C07305=1204.905,265.539,-64.446,-176.922,6.908,148.380
C07306=1204.909,265.290,-64.417,-176.924,6.905,148.380
C07307=1204.914,265.042,-64.390,-176.927,6.904,148.381
C07308=1204.918,264.794,-64.363,-176.929,6.901,148.381
C07309=1204.923,264.545,-64.336,-176.932,6.899,148.381
C07310=1204.926,264.297,-64.307,-176.935,6.896,148.381
C07311=1204.931,264.048,-64.280,-176.937,6.893,148.381
C07312=1204.936,263.800,-64.253,-176.939,6.892,148.382
C07313=1204.939,263.551,-64.225,-176.942,6.889,148.382
C07314=1204.945,263.279,-64.195,-176.945,6.887,148.382
C07315=1204.949,263.006,-64.165,-176.947,6.884,148.382
C07316=1204.954,262.734,-64.135,-176.951,6.881,148.382
C07317=1204.959,262.460,-64.105,-176.953,6.879,148.382
C07318=1204.964,262.212,-64.077,-176.956,6.876,148.383
C07319=1204.968,261.963,-64.050,-176.958,6.874,148.383
C07320=1204.972,261.715,-64.024,-176.961,6.872,148.383
C07321=1204.976,261.467,-63.995,-176.963,6.869,148.383
C07322=1204.981,261.218,-63.968,-176.966,6.867,148.383
C07323=1204.985,260.970,-63.941,-176.968,6.865,148.383
C07324=1204.990,260.721,-63.914,-176.971,6.862,148.384
C07325=1204.994,260.473,-63.886,-176.973,6.860,148.384
C07326=1204.999,260.224,-63.859,-176.977,6.858,148.384
C07327=1205.003,259.976,-63.832,-176.979,6.855,148.384
C07328=1205.008,259.727,-63.805,-176.981,6.853,148.384
C07329=1205.012,259.479,-63.777,-176.984,6.850,148.384
C07330=1205.017,259.231,-63.750,-176.986,6.848,148.384
C07331=1205.021,258.982,-63.723,-176.989,6.846,148.385
C07332=1205.026,258.733,-63.696,-176.992,6.843,148.385
C07333=1205.029,258.485,-63.669,-176.994,6.842,148.385
C07334=1205.034,258.236,-63.642,-176.996,6.839,148.385
C07335=1205.039,257.988,-63.615,-176.999,6.838,148.386
C07336=1205.043,257.740,-63.587,-177.002,6.835,148.386
C07337=1205.047,257.491,-63.560,-177.004,6.833,148.386
C07338=1205.052,257.242,-63.533,-177.006,6.830,148.386
C07339=1205.057,256.994,-63.506,-177.010,6.828,148.386
C07340=1205.060,256.746,-63.479,-177.012,6.826,148.386
C07341=1205.065,256.497,-63.452,-177.014,6.824,148.387
C07342=1205.070,256.249,-63.425,-177.017,6.821,148.387
C07343=1205.074,256.000,-63.398,-177.020,6.819,148.387
C07344=1205.079,255.752,-63.371,-177.022,6.817,148.387
C07345=1205.082,255.503,-63.344,-177.025,6.814,148.387
C07346=1205.087,255.254,-63.317,-177.027,6.812,148.387
C07347=1205.092,255.006,-63.290,-177.030,6.810,148.388
C07348=1205.096,254.757,-63.263,-177.032,6.807,148.388
C07349=1205.100,254.509,-63.236,-177.035,6.805,148.388
C07350=1205.105,254.261,-63.209,-177.037,6.803,148.388
C07351=1205.110,254.012,-63.182,-177.040,6.801,148.389
C07352=1205.114,253.764,-63.155,-177.043,6.798,148.389
C07353=1205.118,253.515,-63.129,-177.045,6.796,148.389
C07354=1205.123,253.267,-63.102,-177.047,6.794,148.389
C07355=1205.127,253.018,-63.075,-177.051,6.791,148.389
C07356=1205.131,252.769,-63.049,-177.053,6.789,148.389
C07357=1205.136,252.520,-63.022,-177.055,6.787,148.390
C07358=1205.140,252.272,-62.994,-177.057,6.785,148.390
C07359=1205.144,252.024,-62.968,-177.061,6.782,148.390
C07360=1205.149,251.775,-62.941,-177.063,6.780,148.390
C07361=1205.154,251.527,-62.914,-177.065,6.778,148.390
C07362=1205.158,251.278,-62.888,-177.069,6.776,148.391
C07363=1205.163,251.029,-62.861,-177.071,6.774,148.391
C07364=1205.167,250.781,-62.834,-177.073,6.772,148.391
C07365=1205.171,250.533,-62.808,-177.076,6.770,148.391
C07366=1205.176,250.284,-62.780,-177.079,6.767,148.391
C07367=1205.181,250.035,-62.754,-177.081,6.765,148.392
C07368=1205.185,249.787,-62.728,-177.083,6.763,148.392
C07369=1205.189,249.539,-62.701,-177.086,6.761,148.392
C07370=1205.193,249.290,-62.674,-177.089,6.758,148.392
C07371=1205.198,249.041,-62.648,-177.091,6.756,148.392
C07372=1205.203,248.793,-62.621,-177.094,6.754,148.393
C07373=1205.207,248.545,-62.594,-177.097,6.751,148.393
C07374=1205.212,248.295,-62.568,-177.099,6.749,148.393
C07375=1205.216,248.047,-62.541,-177.102,6.747,148.393
C07376=1205.220,247.799,-62.514,-177.104,6.745,148.393
C07377=1205.224,247.550,-62.489,-177.107,6.742,148.394
C07378=1205.229,247.301,-62.462,-177.109,6.740,148.394
C07379=1205.233,247.053,-62.436,-177.112,6.738,148.394
C07380=1205.238,246.804,-62.409,-177.114,6.737,148.394
C07381=1205.242,246.556,-62.382,-177.117,6.733,148.394
C07382=1205.248,246.308,-62.356,-177.120,6.732,148.395
C07383=1205.251,246.059,-62.330,-177.122,6.729,148.395
C07384=1205.256,245.810,-62.304,-177.124,6.728,148.395
C07385=1205.260,245.562,-62.277,-177.128,6.725,148.395
C07386=1205.265,245.313,-62.251,-177.130,6.723,148.395
C07387=1205.269,245.065,-62.224,-177.132,6.721,148.396
C07388=1205.274,244.816,-62.198,-177.135,6.719,148.396
C07389=1205.278,244.567,-62.171,-177.137,6.717,148.396
C07390=1205.283,244.318,-62.145,-177.140,6.714,148.396
C07391=1205.287,244.070,-62.119,-177.142,6.712,148.397
C07392=1205.291,243.821,-62.093,-177.145,6.710,148.397
C07393=1205.296,243.573,-62.066,-177.147,6.708,148.397
C07394=1205.301,243.325,-62.040,-177.150,6.705,148.397
C07395=1205.305,243.076,-62.013,-177.153,6.703,148.398
C07396=1205.310,242.827,-61.988,-177.155,6.701,148.398
C07397=1205.314,242.579,-61.962,-177.158,6.699,148.398
C07398=1205.318,242.330,-61.935,-177.160,6.697,148.398
C07399=1205.323,242.081,-61.909,-177.163,6.695,148.398
C07400=1205.327,241.833,-61.883,-177.166,6.693,148.399
C07401=1205.332,241.585,-61.857,-177.168,6.691,148.399
C07402=1205.336,241.336,-61.831,-177.171,6.689,148.399
C07403=1205.341,241.087,-61.804,-177.174,6.686,148.399
C07404=1205.345,240.839,-61.778,-177.176,6.684,148.399
C07405=1205.349,240.590,-61.752,-177.179,6.682,148.400
C07406=1205.354,240.341,-61.725,-177.181,6.680,148.400
C07407=1205.359,240.093,-61.700,-177.183,6.678,148.400
C07408=1205.363,239.844,-61.674,-177.187,6.675,148.400
C07409=1205.367,239.596,-61.648,-177.189,6.673,148.401
C07410=1205.372,239.347,-61.621,-177.191,6.671,148.401
C07411=1205.376,239.098,-61.596,-177.194,6.669,148.401
C07412=1205.381,238.850,-61.570,-177.196,6.667,148.401
C07413=1205.386,238.601,-61.544,-177.199,6.665,148.402
C07414=1205.390,238.353,-61.517,-177.202,6.663,148.402
C07415=1205.394,238.104,-61.492,-177.204,6.661,148.402
C07416=1205.398,237.855,-61.466,-177.207,6.659,148.402
C07417=1205.403,237.607,-61.440,-177.209,6.657,148.403
C07418=1205.408,237.336,-61.411,-177.212,6.654,148.403
C07419=1205.413,237.064,-61.383,-177.215,6.652,148.403
C07420=1205.418,236.793,-61.355,-177.218,6.649,148.403
C07421=1205.423,236.521,-61.327,-177.220,6.648,148.404
C07422=1205.427,236.272,-61.301,-177.223,6.645,148.404
C07423=1205.431,236.024,-61.275,-177.226,6.643,148.404
C07424=1205.437,235.775,-61.249,-177.228,6.641,148.404
C07425=1205.441,235.526,-61.223,-177.231,6.639,148.404
C07426=1205.445,235.278,-61.198,-177.233,6.637,148.405
C07427=1205.450,235.029,-61.172,-177.236,6.635,148.405
C07428=1205.454,234.781,-61.146,-177.239,6.633,148.405
C07429=1205.458,234.532,-61.121,-177.241,6.630,148.405
C07430=1205.463,234.283,-61.095,-177.244,6.628,148.406
C07431=1205.468,234.035,-61.069,-177.247,6.626,148.406
C07432=1205.473,233.786,-61.043,-177.249,6.624,148.406
C07433=1205.477,233.537,-61.018,-177.251,6.622,148.407
C07434=1205.482,233.289,-60.992,-177.254,6.621,148.407
C07435=1205.486,233.040,-60.966,-177.257,6.618,148.407
C07436=1205.490,232.791,-60.941,-177.259,6.616,148.407
C07437=1205.494,232.543,-60.915,-177.262,6.614,148.408
C07438=1205.499,232.294,-60.889,-177.264,6.612,148.408
C07439=1205.503,232.046,-60.864,-177.267,6.610,148.408
C07440=1205.508,231.797,-60.838,-177.269,6.608,148.408
C07441=1205.512,231.549,-60.813,-177.273,6.605,148.409
C07442=1205.517,231.300,-60.787,-177.275,6.603,148.409
C07443=1205.521,231.051,-60.761,-177.277,6.601,148.409
C07444=1205.526,230.802,-60.736,-177.280,6.600,148.409
C07445=1205.531,230.553,-60.710,-177.282,6.597,148.409
C07446=1205.536,230.305,-60.685,-177.285,6.596,148.410
C07447=1205.540,230.056,-60.659,-177.287,6.594,148.410
C07448=1205.544,229.808,-60.633,-177.291,6.591,148.410
C07449=1205.548,229.560,-60.608,-177.293,6.589,148.410
C07450=1205.553,229.310,-60.583,-177.295,6.587,148.411
C07451=1205.557,229.062,-60.558,-177.298,6.585,148.411
C07452=1205.562,228.813,-60.532,-177.301,6.583,148.411
C07453=1205.566,228.565,-60.506,-177.303,6.581,148.412
C07454=1205.571,228.316,-60.482,-177.305,6.579,148.412
C07455=1205.575,228.067,-60.456,-177.308,6.577,148.412
C07456=1205.580,227.818,-60.430,-177.311,6.575,148.413
C07457=1205.584,227.570,-60.405,-177.313,6.573,148.413
C07458=1205.589,227.321,-60.380,-177.316,6.571,148.413
C07459=1205.594,227.073,-60.355,-177.319,6.569,148.413
C07460=1205.598,226.824,-60.329,-177.321,6.567,148.414
C07461=1205.603,226.575,-60.304,-177.323,6.565,148.414
C07462=1205.607,226.326,-60.278,-177.326,6.563,148.414
C07463=1205.612,226.078,-60.253,-177.329,6.560,148.414
C07464=1205.616,225.829,-60.229,-177.332,6.559,148.415
C07465=1205.620,225.580,-60.203,-177.334,6.556,148.415
C07466=1205.625,225.332,-60.178,-177.337,6.555,148.415
C07467=1205.630,225.083,-60.152,-177.339,6.553,148.415
C07468=1205.634,224.835,-60.127,-177.342,6.551,148.416
C07469=1205.639,224.585,-60.102,-177.344,6.549,148.416
C07470=1205.643,224.337,-60.077,-177.347,6.547,148.416
C07471=1205.648,224.088,-60.052,-177.349,6.545,148.417
C07472=1205.652,223.840,-60.027,-177.353,6.542,148.417
C07473=1205.657,223.591,-60.002,-177.355,6.540,148.417
C07474=1205.662,223.342,-59.976,-177.357,6.538,148.417
C07475=1205.666,223.093,-59.951,-177.360,6.537,148.418
C07476=1205.670,222.845,-59.926,-177.363,6.535,148.418
C07477=1205.675,222.596,-59.901,-177.365,6.533,148.418
C07478=1205.680,222.348,-59.876,-177.368,6.531,148.418
C07479=1205.684,222.098,-59.851,-177.370,6.529,148.419
C07480=1205.688,221.850,-59.826,-177.373,6.527,148.419
C07481=1205.693,221.601,-59.801,-177.375,6.525,148.419
C07482=1205.698,221.353,-59.776,-177.379,6.523,148.420
C07483=1205.702,221.103,-59.751,-177.381,6.520,148.420
C07484=1205.706,220.856,-59.726,-177.383,6.519,148.420
C07485=1205.711,220.606,-59.701,-177.386,6.517,148.420
C07486=1205.716,220.358,-59.676,-177.389,6.515,148.421
C07487=1205.719,220.109,-59.651,-177.391,6.513,148.421
C07488=1205.725,219.860,-59.626,-177.393,6.511,148.421
C07489=1205.729,219.611,-59.601,-177.396,6.509,148.421
C07490=1205.733,219.363,-59.577,-177.399,6.507,148.422
C07491=1205.738,219.114,-59.552,-177.401,6.505,148.422
C07492=1205.743,218.865,-59.527,-177.405,6.503,148.422
C07493=1205.747,218.617,-59.502,-177.407,6.501,148.423
C07494=1205.752,218.368,-59.477,-177.409,6.499,148.423
C07495=1205.757,218.119,-59.452,-177.412,6.497,148.423
C07496=1205.760,217.871,-59.427,-177.415,6.495,148.424
C07497=1205.765,217.622,-59.403,-177.417,6.493,148.424
C07498=1205.770,217.373,-59.378,-177.420,6.491,148.424
C07499=1205.774,217.124,-59.353,-177.423,6.489,148.425
C07500=1205.779,216.876,-59.328,-177.425,6.487,148.425
C07501=1205.783,216.627,-59.304,-177.427,6.485,148.425
C07502=1205.788,216.378,-59.279,-177.430,6.484,148.425
C07503=1205.793,216.129,-59.254,-177.433,6.482,148.426
C07504=1205.797,215.880,-59.230,-177.435,6.480,148.426
C07505=1205.802,215.632,-59.204,-177.439,6.477,148.426
C07506=1205.806,215.384,-59.180,-177.441,6.475,148.426
C07507=1205.811,215.134,-59.155,-177.443,6.473,148.427
C07508=1205.815,214.886,-59.131,-177.446,6.471,148.427
C07509=1205.820,214.636,-59.106,-177.449,6.470,148.427
C07510=1205.824,214.388,-59.082,-177.451,6.468,148.428
C07511=1205.829,214.139,-59.058,-177.454,6.466,148.428
C07512=1205.833,213.890,-59.033,-177.457,6.464,148.428
C07513=1205.838,213.642,-59.008,-177.459,6.462,148.429
C07514=1205.842,213.394,-58.984,-177.461,6.460,148.429
C07515=1205.847,213.144,-58.959,-177.464,6.458,148.429
C07516=1205.851,212.896,-58.935,-177.467,6.456,148.430
C07517=1205.856,212.647,-58.910,-177.469,6.455,148.430
C07518=1205.861,212.399,-58.886,-177.472,6.453,148.430
C07519=1205.865,212.149,-58.861,-177.475,6.451,148.431
C07520=1205.869,211.901,-58.837,-177.477,6.449,148.431
C07521=1205.875,211.652,-58.812,-177.480,6.446,148.431
C07522=1205.879,211.381,-58.785,-177.483,6.444,148.431
C07523=1205.884,211.111,-58.760,-177.485,6.443,148.432
C07524=1205.889,210.841,-58.733,-177.488,6.441,148.432
C07525=1205.894,210.570,-58.706,-177.492,6.438,148.432
C07526=1205.898,210.321,-58.682,-177.494,6.436,148.433
C07527=1205.903,210.073,-58.657,-177.496,6.434,148.433
C07528=1205.907,209.824,-58.633,-177.499,6.433,148.433
C07529=1205.913,209.575,-58.608,-177.502,6.431,148.434
C07530=1205.917,209.326,-58.585,-177.504,6.429,148.434
C07531=1205.921,209.077,-58.560,-177.507,6.427,148.434
C07532=1205.926,208.829,-58.536,-177.510,6.425,148.435
C07533=1205.931,208.580,-58.512,-177.512,6.423,148.435
C07534=1205.935,208.332,-58.488,-177.515,6.422,148.435
C07535=1205.940,208.082,-58.463,-177.518,6.420,148.436
C07536=1205.944,207.834,-58.439,-177.520,6.418,148.436
C07537=1205.949,207.585,-58.415,-177.522,6.416,148.436
C07538=1205.954,207.336,-58.390,-177.525,6.414,148.436
C07539=1205.958,207.087,-58.366,-177.528,6.412,148.437
C07540=1205.962,206.839,-58.342,-177.530,6.410,148.437
C07541=1205.967,206.589,-58.318,-177.533,6.408,148.437
C07542=1205.972,206.341,-58.294,-177.536,6.407,148.438
C07543=1205.976,206.092,-58.270,-177.538,6.405,148.438
C07544=1205.981,205.843,-58.245,-177.541,6.403,148.438
C07545=1205.985,205.594,-58.221,-177.544,6.401,148.439
C07546=1205.990,205.346,-58.197,-177.546,6.399,148.439
C07547=1205.994,205.097,-58.173,-177.548,6.397,148.439
C07548=1205.999,204.848,-58.149,-177.551,6.395,148.440
C07549=1206.004,204.599,-58.125,-177.554,6.393,148.440
C07550=1206.008,204.350,-58.101,-177.556,6.392,148.440
C07551=1206.012,204.102,-58.077,-177.559,6.390,148.441
C07552=1206.017,203.853,-58.053,-177.562,6.388,148.441
C07553=1206.022,203.604,-58.029,-177.564,6.386,148.441
C07554=1206.027,203.355,-58.005,-177.567,6.384,148.442
C07555=1206.031,203.107,-57.981,-177.570,6.382,148.442
C07556=1206.036,202.858,-57.957,-177.572,6.381,148.442
C07557=1206.040,202.609,-57.934,-177.575,6.379,148.443
C07558=1206.045,202.360,-57.909,-177.577,6.377,148.443
C07559=1206.049,202.111,-57.885,-177.580,6.375,148.443
C07560=1206.054,201.862,-57.861,-177.583,6.373,148.444
C07561=1206.058,201.614,-57.837,-177.585,6.372,148.444
C07562=1206.063,201.365,-57.814,-177.588,6.369,148.444
C07563=1206.067,201.117,-57.790,-177.590,6.368,148.444
C07564=1206.072,200.868,-57.767,-177.593,6.366,148.445
C07565=1206.077,200.619,-57.742,-177.596,6.364,148.445
C07566=1206.081,200.369,-57.718,-177.598,6.362,148.446
C07567=1206.086,200.121,-57.694,-177.601,6.360,148.446
C07568=1206.090,199.872,-57.671,-177.603,6.358,148.446
C07569=1206.095,199.623,-57.647,-177.606,6.357,148.447
C07570=1206.099,199.374,-57.623,-177.609,6.355,148.447
C07571=1206.104,199.125,-57.600,-177.611,6.353,148.447
C07572=1206.109,198.877,-57.576,-177.614,6.351,148.448
C07573=1206.113,198.628,-57.552,-177.617,6.349,148.448
C07574=1206.118,198.379,-57.528,-177.619,6.347,148.448
C07575=1206.122,198.130,-57.505,-177.622,6.346,148.449
C07576=1206.127,197.881,-57.482,-177.625,6.344,148.449
C07577=1206.131,197.633,-57.458,-177.627,6.342,148.449
C07578=1206.136,197.384,-57.434,-177.629,6.341,148.450
C07579=1206.141,197.135,-57.411,-177.632,6.339,148.450
C07580=1206.145,196.886,-57.387,-177.635,6.337,148.450
C07581=1206.150,196.637,-57.363,-177.637,6.336,148.451
C07582=1206.155,196.388,-57.340,-177.640,6.334,148.451
C07583=1206.159,196.140,-57.316,-177.643,6.332,148.451
C07584=1206.164,195.891,-57.293,-177.645,6.330,148.452
C07585=1206.168,195.642,-57.269,-177.648,6.328,148.452
C07586=1206.173,195.393,-57.245,-177.651,6.326,148.452
C07587=1206.178,195.144,-57.222,-177.653,6.325,148.453
C07588=1206.182,194.895,-57.199,-177.656,6.323,148.453
C07589=1206.187,194.646,-57.175,-177.659,6.321,148.453
C07590=1206.191,194.398,-57.151,-177.661,6.319,148.454
C07591=1206.196,194.149,-57.128,-177.664,6.317,148.454
C07592=1206.201,193.900,-57.104,-177.667,6.316,148.455
C07593=1206.205,193.651,-57.081,-177.669,6.314,148.455
C07594=1206.210,193.402,-57.058,-177.671,6.313,148.455
C07595=1206.215,193.153,-57.034,-177.674,6.311,148.456
C07596=1206.219,192.904,-57.010,-177.677,6.309,148.456
C07597=1206.223,192.656,-56.987,-177.679,6.307,148.456
C07598=1206.228,192.407,-56.964,-177.682,6.305,148.457
C07599=1206.233,192.157,-56.941,-177.685,6.304,148.457
C07600=1206.237,191.908,-56.917,-177.687,6.302,148.457
C07601=1206.242,191.659,-56.894,-177.690,6.300,148.458
C07602=1206.247,191.410,-56.871,-177.693,6.298,148.458
C07603=1206.252,191.163,-56.847,-177.695,6.296,148.458
C07604=1206.256,190.914,-56.824,-177.698,6.295,148.459
C07605=1206.260,190.665,-56.801,-177.700,6.293,148.459
C07606=1206.265,190.416,-56.777,-177.703,6.292,148.459
C07607=1206.270,190.167,-56.754,-177.705,6.290,148.460
C07608=1206.274,189.918,-56.731,-177.708,6.288,148.460
C07609=1206.279,189.669,-56.707,-177.711,6.286,148.461
C07610=1206.283,189.420,-56.685,-177.713,6.284,148.461
C07611=1206.288,189.171,-56.661,-177.716,6.283,148.461
C07612=1206.293,188.923,-56.638,-177.718,6.281,148.462
C07613=1206.298,188.674,-56.615,-177.721,6.279,148.462
C07614=1206.302,188.425,-56.592,-177.724,6.277,148.462
C07615=1206.306,188.176,-56.569,-177.726,6.276,148.463
C07616=1206.311,187.927,-56.545,-177.729,6.274,148.463
C07617=1206.316,187.678,-56.522,-177.731,6.273,148.463
C07618=1206.320,187.429,-56.499,-177.734,6.271,148.464
C07619=1206.325,187.181,-56.476,-177.737,6.269,148.464
C07620=1206.330,186.931,-56.454,-177.739,6.267,148.464
C07621=1206.335,186.682,-56.430,-177.742,6.265,148.465
C07622=1206.339,186.433,-56.408,-177.744,6.263,148.465
C07623=1206.343,186.184,-56.384,-177.747,6.262,148.465
C07624=1206.348,185.935,-56.361,-177.749,6.261,148.466
C07625=1206.353,185.687,-56.338,-177.752,6.259,148.466
C07626=1206.358,185.418,-56.313,-177.755,6.257,148.467
C07627=1206.363,185.148,-56.288,-177.758,6.256,148.467
C07628=1206.368,184.878,-56.264,-177.761,6.253,148.467
C07629=1206.373,184.609,-56.239,-177.764,6.251,148.468
C07630=1206.377,184.360,-56.216,-177.766,6.249,148.468
C07631=1206.382,184.111,-56.193,-177.768,6.248,148.469
C07632=1206.387,183.861,-56.170,-177.771,6.246,148.469
C07633=1206.391,183.612,-56.147,-177.774,6.245,148.469
C07634=1206.396,183.364,-56.124,-177.777,6.243,148.470
C07635=1206.401,183.115,-56.101,-177.779,6.241,148.470
C07636=1206.405,182.866,-56.079,-177.782,6.240,148.471
C07637=1206.410,182.617,-56.056,-177.785,6.238,148.471
C07638=1206.414,182.368,-56.033,-177.787,6.237,148.471
C07639=1206.419,182.120,-56.010,-177.790,6.235,148.472
C07640=1206.423,181.870,-55.988,-177.792,6.233,148.472
C07641=1206.428,181.621,-55.964,-177.795,6.231,148.472
C07642=1206.433,181.372,-55.941,-177.797,6.229,148.473
C07643=1206.438,181.124,-55.919,-177.800,6.228,148.473
C07644=1206.442,180.875,-55.896,-177.802,6.227,148.473
C07645=1206.446,180.626,-55.873,-177.805,6.225,148.474
C07646=1206.452,180.377,-55.851,-177.808,6.223,148.474
C07647=1206.456,180.128,-55.828,-177.811,6.222,148.475
C07648=1206.461,179.879,-55.806,-177.813,6.220,148.475
C07649=1206.465,179.630,-55.783,-177.816,6.218,148.475
C07650=1206.470,179.381,-55.760,-177.818,6.217,148.476
C07651=1206.474,179.132,-55.738,-177.821,6.215,148.476
C07652=1206.479,178.883,-55.714,-177.823,6.213,148.477
C07653=1206.484,178.634,-55.693,-177.826,6.212,148.477
C07654=1206.489,178.385,-55.669,-177.829,6.210,148.477
C07655=1206.493,178.136,-55.647,-177.831,6.208,148.478
C07656=1206.498,177.888,-55.624,-177.834,6.207,148.478
C07657=1206.503,177.638,-55.602,-177.837,6.205,148.479
C07658=1206.507,177.390,-55.580,-177.839,6.204,148.479
C07659=1206.512,177.141,-55.557,-177.842,6.202,148.479
C07660=1206.516,176.892,-55.535,-177.845,6.200,148.480
C07661=1206.521,176.642,-55.512,-177.847,6.198,148.480
C07662=1206.526,176.394,-55.489,-177.849,6.197,148.480
C07663=1206.531,176.145,-55.467,-177.852,6.195,148.481
C07664=1206.535,175.896,-55.444,-177.855,6.194,148.481
C07665=1206.540,175.647,-55.422,-177.857,6.192,148.481
C07666=1206.545,175.398,-55.400,-177.861,6.190,148.482
C07667=1206.548,175.149,-55.377,-177.863,6.189,148.482
C07668=1206.554,174.900,-55.355,-177.865,6.188,148.483
C07669=1206.558,174.651,-55.332,-177.868,6.186,148.483
C07670=1206.563,174.403,-55.310,-177.871,6.184,148.484
C07671=1206.568,174.153,-55.288,-177.873,6.182,148.484
C07672=1206.572,173.904,-55.265,-177.875,6.181,148.484
C07673=1206.577,173.656,-55.243,-177.878,6.179,148.485
C07674=1206.582,173.406,-55.221,-177.881,6.178,148.485
C07675=1206.586,173.158,-55.198,-177.884,6.176,148.486
C07676=1206.591,172.909,-55.176,-177.887,6.174,148.486
C07677=1206.596,172.659,-55.153,-177.889,6.173,148.486
C07678=1206.600,172.411,-55.131,-177.891,6.171,148.487
C07679=1206.604,172.162,-55.109,-177.894,6.170,148.487
C07680=1206.609,171.913,-55.087,-177.897,6.168,148.487
C07681=1206.614,171.663,-55.065,-177.899,6.167,148.488
C07682=1206.619,171.415,-55.042,-177.902,6.165,148.488
C07683=1206.623,171.166,-55.020,-177.905,6.164,148.489
C07684=1206.628,170.916,-54.998,-177.907,6.162,148.489
C07685=1206.633,170.668,-54.976,-177.910,6.160,148.489
C07686=1206.637,170.418,-54.954,-177.912,6.159,148.490
C07687=1206.642,170.170,-54.931,-177.915,6.157,148.490
C07688=1206.647,169.921,-54.909,-177.918,6.156,148.491
C07689=1206.652,169.672,-54.887,-177.920,6.154,148.491
C07690=1206.656,169.423,-54.865,-177.923,6.153,148.492
C07691=1206.661,169.174,-54.843,-177.925,6.151,148.492
C07692=1206.665,168.925,-54.821,-177.928,6.149,148.492
C07693=1206.670,168.676,-54.798,-177.931,6.148,148.493
C07694=1206.675,168.427,-54.776,-177.933,6.147,148.493
C07695=1206.680,168.178,-54.755,-177.936,6.145,148.494
C07696=1206.684,167.929,-54.733,-177.938,6.143,148.494
C07697=1206.689,167.680,-54.711,-177.941,6.141,148.494
C07698=1206.693,167.431,-54.689,-177.943,6.140,148.495
C07699=1206.699,167.182,-54.667,-177.946,6.139,148.495
C07700=1206.703,166.933,-54.644,-177.949,6.137,148.495
C07701=1206.708,166.684,-54.623,-177.952,6.135,148.496
C07702=1206.712,166.435,-54.601,-177.954,6.134,148.496
C07703=1206.717,166.186,-54.579,-177.956,6.133,148.497
C07704=1206.721,165.937,-54.557,-177.959,6.131,148.497
C07705=1206.726,165.688,-54.535,-177.962,6.129,148.498
C07706=1206.730,165.439,-54.513,-177.964,6.128,148.498
C07707=1206.736,165.190,-54.491,-177.967,6.127,148.499
C07708=1206.741,164.941,-54.469,-177.970,6.125,148.499
C07709=1206.745,164.692,-54.447,-177.972,6.123,148.499
C07710=1206.750,164.443,-54.426,-177.975,6.122,148.500
C07711=1206.754,164.194,-54.404,-177.977,6.120,148.500
C07712=1206.759,163.945,-54.382,-177.980,6.119,148.501
C07713=1206.763,163.696,-54.360,-177.982,6.118,148.501
C07714=1206.768,163.447,-54.338,-177.985,6.116,148.501
C07715=1206.773,163.199,-54.316,-177.988,6.114,148.502
C07716=1206.777,162.949,-54.294,-177.990,6.112,148.502
C07717=1206.782,162.701,-54.273,-177.993,6.112,148.503
C07718=1206.787,162.451,-54.251,-177.996,6.110,148.503
C07719=1206.792,162.202,-54.230,-177.998,6.108,148.503
C07720=1206.796,161.953,-54.208,-178.001,6.106,148.504
C07721=1206.801,161.704,-54.186,-178.003,6.105,148.504
C07722=1206.806,161.455,-54.164,-178.006,6.104,148.505
C07723=1206.810,161.206,-54.142,-178.009,6.102,148.505
C07724=1206.815,160.957,-54.121,-178.011,6.101,148.506
C07725=1206.820,160.708,-54.100,-178.014,6.099,148.506
C07726=1206.824,160.459,-54.078,-178.017,6.098,148.507
C07727=1206.829,160.210,-54.056,-178.020,6.096,148.507
C07728=1206.834,159.961,-54.035,-178.022,6.095,148.507
C07729=1206.838,159.712,-54.013,-178.024,6.093,148.508
C07730=1206.843,159.443,-53.989,-178.027,6.092,148.508
C07731=1206.848,159.174,-53.966,-178.030,6.090,148.509
C07732=1206.853,158.905,-53.943,-178.033,6.088,148.509
C07733=1206.859,158.635,-53.920,-178.036,6.087,148.510
C07734=1206.864,158.387,-53.898,-178.038,6.086,148.510
C07735=1206.868,158.138,-53.877,-178.041,6.084,148.510
C07736=1206.873,157.889,-53.854,-178.043,6.082,148.511
C07737=1206.878,157.640,-53.834,-178.046,6.082,148.511
C07738=1206.882,157.391,-53.812,-178.049,6.080,148.512
C07739=1206.886,157.142,-53.790,-178.051,6.078,148.512
C07740=1206.891,156.893,-53.769,-178.053,6.077,148.512
C07741=1206.896,156.644,-53.748,-178.057,6.076,148.513
C07742=1206.901,156.394,-53.726,-178.059,6.074,148.513
C07743=1206.906,156.145,-53.705,-178.061,6.073,148.514
C07744=1206.911,155.897,-53.683,-178.064,6.071,148.514
C07745=1206.915,155.648,-53.663,-178.067,6.069,148.515
C07746=1206.919,155.398,-53.641,-178.069,6.069,148.515
C07747=1206.924,155.149,-53.620,-178.072,6.067,148.516
C07748=1206.929,154.901,-53.598,-178.075,6.065,148.516
C07749=1206.934,154.651,-53.577,-178.077,6.064,148.517
C07750=1206.938,154.402,-53.556,-178.080,6.063,148.517
C07751=1206.943,154.153,-53.535,-178.083,6.061,148.517
C07752=1206.948,153.904,-53.513,-178.085,6.060,148.518
C07753=1206.953,153.656,-53.491,-178.088,6.058,148.518
C07754=1206.958,153.406,-53.470,-178.091,6.056,148.519
C07755=1206.962,153.157,-53.450,-178.093,6.056,148.519
C07756=1206.967,152.908,-53.428,-178.095,6.054,148.519
C07757=1206.972,152.659,-53.407,-178.099,6.052,148.520
C07758=1206.976,152.410,-53.385,-178.101,6.051,148.520
C07759=1206.981,152.161,-53.364,-178.103,6.050,148.521
C07760=1206.986,151.912,-53.343,-178.106,6.048,148.521
C07761=1206.991,151.663,-53.322,-178.109,6.047,148.522
C07762=1206.996,151.414,-53.300,-178.111,6.045,148.522
C07763=1206.999,151.164,-53.279,-178.114,6.044,148.523
C07764=1207.005,150.915,-53.258,-178.116,6.043,148.523
C07765=1207.009,150.667,-53.237,-178.119,6.041,148.524
C07766=1207.014,150.418,-53.216,-178.122,6.039,148.524
C07767=1207.019,150.169,-53.195,-178.124,6.038,148.524
C07768=1207.023,149.919,-53.173,-178.127,6.037,148.525
C07769=1207.028,149.670,-53.153,-178.129,6.036,148.525
C07770=1207.033,149.421,-53.131,-178.132,6.034,148.526
C07771=1207.038,149.172,-53.110,-178.135,6.032,148.526
C07772=1207.042,148.923,-53.090,-178.137,6.032,148.527
C07773=1207.047,148.674,-53.069,-178.140,6.030,148.527
C07774=1207.052,148.425,-53.047,-178.143,6.028,148.527
C07775=1207.056,148.176,-53.027,-178.145,6.027,148.528
C07776=1207.061,147.926,-53.006,-178.148,6.026,148.528
C07777=1207.065,147.678,-52.985,-178.150,6.024,148.529
C07778=1207.071,147.429,-52.964,-178.153,6.023,148.529
C07779=1207.076,147.180,-52.943,-178.156,6.021,148.530
C07780=1207.080,146.931,-52.922,-178.158,6.021,148.530
C07781=1207.085,146.681,-52.900,-178.161,6.019,148.531
C07782=1207.089,146.432,-52.880,-178.164,6.017,148.531
C07783=1207.094,146.183,-52.859,-178.166,6.016,148.532
C07784=1207.099,145.934,-52.838,-178.168,6.015,148.532
C07785=1207.104,145.685,-52.817,-178.171,6.014,148.533
C07786=1207.109,145.436,-52.796,-178.174,6.012,148.533
C07787=1207.113,145.187,-52.775,-178.176,6.010,148.533
C07788=1207.118,144.938,-52.754,-178.179,6.010,148.534
C07789=1207.123,144.689,-52.734,-178.182,6.008,148.534
C07790=1207.127,144.439,-52.713,-178.184,6.007,148.535
C07791=1207.132,144.190,-52.692,-178.186,6.005,148.535
C07792=1207.137,143.941,-52.671,-178.190,6.004,148.536
C07793=1207.141,143.692,-52.651,-178.192,6.003,148.536
C07794=1207.146,143.443,-52.629,-178.194,6.001,148.537
C07795=1207.151,143.194,-52.609,-178.197,6.000,148.537
C07796=1207.156,142.945,-52.588,-178.200,5.999,148.538
C07797=1207.160,142.696,-52.568,-178.202,5.997,148.538
C07798=1207.165,142.447,-52.547,-178.205,5.996,148.539
C07799=1207.170,142.198,-52.526,-178.208,5.994,148.539
C07800=1207.174,141.949,-52.506,-178.210,5.993,148.539
C07801=1207.179,141.700,-52.485,-178.213,5.992,148.540
C07802=1207.184,141.451,-52.465,-178.216,5.990,148.540
C07803=1207.189,141.201,-52.444,-178.218,5.989,148.541
C07804=1207.193,140.953,-52.423,-178.221,5.988,148.541
C07805=1207.199,140.703,-52.402,-178.223,5.987,148.542
C07806=1207.203,140.454,-52.382,-178.226,5.985,148.542
C07807=1207.208,140.205,-52.362,-178.228,5.984,148.543
C07808=1207.213,139.956,-52.341,-178.231,5.983,148.543
C07809=1207.217,139.707,-52.320,-178.234,5.981,148.544
C07810=1207.222,139.458,-52.300,-178.236,5.980,148.544
C07811=1207.227,139.209,-52.279,-178.239,5.978,148.545
C07812=1207.232,138.959,-52.259,-178.241,5.977,148.545
C07813=1207.237,138.710,-52.238,-178.244,5.976,148.546
C07814=1207.241,138.461,-52.218,-178.246,5.975,148.546
C07815=1207.246,138.212,-52.198,-178.249,5.973,148.546
C07816=1207.251,137.963,-52.177,-178.252,5.972,148.547
C07817=1207.255,137.714,-52.156,-178.254,5.971,148.547
C07818=1207.260,137.465,-52.136,-178.257,5.969,148.548
C07819=1207.265,137.216,-52.115,-178.260,5.968,148.548
C07820=1207.270,136.966,-52.095,-178.262,5.967,148.549
C07821=1207.274,136.717,-52.075,-178.265,5.966,148.549
C07822=1207.279,136.468,-52.054,-178.268,5.964,148.550
C07823=1207.284,136.219,-52.033,-178.270,5.963,148.550
C07824=1207.288,135.970,-52.013,-178.273,5.962,148.551
C07825=1207.293,135.721,-51.993,-178.276,5.960,148.551
C07826=1207.298,135.471,-51.972,-178.278,5.959,148.552
C07827=1207.302,135.222,-51.952,-178.281,5.958,148.552
C07828=1207.307,134.973,-51.932,-178.283,5.957,148.553
C07829=1207.312,134.724,-51.912,-178.286,5.955,148.553
C07830=1207.317,134.475,-51.891,-178.288,5.954,148.554
C07831=1207.322,134.226,-51.871,-178.291,5.953,148.554
C07832=1207.326,133.977,-51.851,-178.293,5.952,148.555
C07833=1207.331,133.728,-51.831,-178.296,5.950,148.555
C07834=1207.336,133.459,-51.809,-178.299,5.949,148.556
C07835=1207.342,133.191,-51.787,-178.301,5.948,148.556
C07836=1207.346,132.922,-51.765,-178.305,5.946,148.557
C07837=1207.352,132.653,-51.743,-178.307,5.945,148.557
C07838=1207.356,132.404,-51.723,-178.310,5.944,148.558
C07839=1207.361,132.155,-51.703,-178.313,5.942,148.558
C07840=1207.366,131.906,-51.683,-178.315,5.941,148.558
C07841=1207.370,131.657,-51.663,-178.318,5.940,148.559
C07842=1207.376,131.407,-51.642,-178.320,5.939,148.559
C07843=1207.380,131.158,-51.622,-178.323,5.937,148.560
C07844=1207.385,130.909,-51.602,-178.325,5.936,148.560
C07845=1207.389,130.660,-51.582,-178.328,5.935,148.561
C07846=1207.394,130.412,-51.562,-178.331,5.934,148.562
C07847=1207.399,130.162,-51.542,-178.333,5.932,148.562
C07848=1207.404,129.913,-51.521,-178.336,5.931,148.562
C07849=1207.409,129.663,-51.502,-178.339,5.930,148.563
C07850=1207.413,129.414,-51.481,-178.341,5.928,148.563
C07851=1207.419,129.165,-51.462,-178.344,5.927,148.564
C07852=1207.423,128.916,-51.442,-178.347,5.926,148.564
C07853=1207.428,128.667,-51.422,-178.349,5.925,148.565
C07854=1207.432,128.418,-51.402,-178.352,5.923,148.565
C07855=1207.437,128.168,-51.382,-178.354,5.922,148.566
C07856=1207.442,127.919,-51.362,-178.357,5.921,148.566
C07857=1207.447,127.670,-51.342,-178.359,5.920,148.567
C07858=1207.451,127.421,-51.322,-178.362,5.919,148.567
C07859=1207.456,127.172,-51.302,-178.365,5.918,148.568
C07860=1207.461,126.923,-51.282,-178.367,5.916,148.568
C07861=1207.465,126.673,-51.262,-178.370,5.915,148.569
C07862=1207.470,126.425,-51.242,-178.372,5.913,148.569
C07863=1207.476,126.175,-51.222,-178.375,5.913,148.570
C07864=1207.481,125.926,-51.202,-178.377,5.912,148.570
C07865=1207.485,125.677,-51.182,-178.380,5.910,148.571
C07866=1207.490,125.428,-51.163,-178.383,5.909,148.571
C07867=1207.495,125.178,-51.143,-178.385,5.908,148.572
C07868=1207.500,124.929,-51.123,-178.388,5.907,148.572
C07869=1207.504,124.680,-51.104,-178.390,5.905,148.573
C07870=1207.509,124.431,-51.084,-178.393,5.905,148.573
C07871=1207.513,124.182,-51.064,-178.396,5.903,148.574
C07872=1207.518,123.933,-51.044,-178.398,5.902,148.574
C07873=1207.523,123.683,-51.025,-178.401,5.901,148.575
C07874=1207.528,123.435,-51.005,-178.403,5.900,148.575
C07875=1207.533,123.185,-50.985,-178.406,5.898,148.576
C07876=1207.537,122.936,-50.965,-178.408,5.897,148.576
C07877=1207.542,122.688,-50.945,-178.412,5.896,148.577
C07878=1207.547,122.438,-50.926,-178.414,5.895,148.577
C07879=1207.552,122.188,-50.906,-178.417,5.893,148.578
C07880=1207.557,121.939,-50.886,-178.419,5.892,148.578
C07881=1207.562,121.691,-50.866,-178.422,5.891,148.579
C07882=1207.566,121.441,-50.847,-178.424,5.890,148.579
C07883=1207.571,121.191,-50.827,-178.427,5.889,148.580
C07884=1207.576,120.943,-50.808,-178.430,5.888,148.580
C07885=1207.580,120.693,-50.789,-178.432,5.887,148.581
C07886=1207.585,120.444,-50.768,-178.435,5.885,148.581
C07887=1207.590,120.196,-50.749,-178.437,5.884,148.582
C07888=1207.595,119.946,-50.729,-178.440,5.883,148.582
C07889=1207.600,119.696,-50.710,-178.442,5.882,148.583
C07890=1207.605,119.448,-50.690,-178.446,5.881,148.583
C07891=1207.609,119.198,-50.671,-178.448,5.880,148.584
C07892=1207.614,118.949,-50.652,-178.450,5.879,148.584
C07893=1207.619,118.700,-50.632,-178.453,5.877,148.585
C07894=1207.624,118.451,-50.612,-178.455,5.876,148.585
C07895=1207.628,118.201,-50.592,-178.458,5.875,148.586
C07896=1207.634,117.952,-50.573,-178.460,5.874,148.586
C07897=1207.638,117.703,-50.554,-178.464,5.873,148.587
C07898=1207.643,117.454,-50.535,-178.466,5.872,148.587
C07899=1207.648,117.205,-50.515,-178.469,5.870,148.588
C07900=1207.653,116.955,-50.496,-178.471,5.869,148.588
C07901=1207.657,116.707,-50.477,-178.474,5.869,148.589
C07902=1207.662,116.457,-50.457,-178.476,5.867,148.589
C07903=1207.667,116.208,-50.438,-178.479,5.866,148.590
C07904=1207.672,115.959,-50.418,-178.482,5.864,148.590
C07905=1207.676,115.709,-50.399,-178.484,5.864,148.591
C07906=1207.681,115.460,-50.380,-178.487,5.862,148.591
C07907=1207.686,115.211,-50.360,-178.490,5.861,148.592
C07908=1207.691,114.962,-50.341,-178.492,5.861,148.593
C07909=1207.695,114.713,-50.322,-178.494,5.859,148.593
C07910=1207.700,114.463,-50.302,-178.497,5.858,148.594
C07911=1207.706,114.214,-50.283,-178.500,5.856,148.594
C07912=1207.710,113.965,-50.263,-178.502,5.856,148.595
C07913=1207.715,113.716,-50.245,-178.504,5.855,148.595
C07914=1207.720,113.467,-50.225,-178.508,5.853,148.596
C07915=1207.725,113.218,-50.206,-178.510,5.852,148.596
C07916=1207.729,112.969,-50.187,-178.513,5.851,148.597
C07917=1207.735,112.719,-50.168,-178.515,5.850,148.597
C07918=1207.739,112.469,-50.148,-178.518,5.849,148.598
C07919=1207.744,112.221,-50.130,-178.520,5.848,148.598
C07920=1207.749,111.971,-50.110,-178.523,5.847,148.599
C07921=1207.753,111.722,-50.090,-178.526,5.845,148.599
C07922=1207.758,111.473,-50.072,-178.528,5.845,148.600
C07923=1207.763,111.224,-50.052,-178.531,5.843,148.600
C07924=1207.768,110.974,-50.034,-178.534,5.842,148.601
C07925=1207.772,110.725,-50.014,-178.536,5.841,148.601
C07926=1207.778,110.476,-49.995,-178.539,5.840,148.602
C07927=1207.782,110.227,-49.976,-178.541,5.839,148.602
C07928=1207.787,109.978,-49.957,-178.544,5.839,148.603
C07929=1207.791,109.728,-49.938,-178.546,5.837,148.603
C07930=1207.797,109.479,-49.919,-178.549,5.836,148.604
C07931=1207.802,109.230,-49.899,-178.552,5.834,148.604
C07932=1207.806,108.981,-49.881,-178.554,5.834,148.605
C07933=1207.811,108.731,-49.862,-178.556,5.833,148.605
C07934=1207.816,108.482,-49.843,-178.560,5.831,148.606
C07935=1207.821,108.233,-49.824,-178.562,5.831,148.607
C07936=1207.825,107.984,-49.805,-178.565,5.829,148.607
C07937=1207.831,107.735,-49.786,-178.567,5.829,148.608
C07938=1207.836,107.466,-49.765,-178.570,5.828,148.608
C07939=1207.841,107.198,-49.746,-178.573,5.826,148.609
C07940=1207.846,106.929,-49.725,-178.576,5.825,148.609
C07941=1207.852,106.661,-49.705,-178.578,5.824,148.610
C07942=1207.856,106.412,-49.686,-178.581,5.823,148.611
C07943=1207.861,106.162,-49.666,-178.583,5.821,148.611
C07944=1207.866,105.913,-49.648,-178.586,5.821,148.612
C07945=1207.871,105.664,-49.629,-178.589,5.819,148.612
C07946=1207.875,105.415,-49.610,-178.591,5.818,148.613
C07947=1207.880,105.165,-49.591,-178.594,5.818,148.613
C07948=1207.885,104.916,-49.572,-178.597,5.816,148.614
C07949=1207.890,104.667,-49.554,-178.599,5.816,148.614
C07950=1207.894,104.418,-49.535,-178.601,5.815,148.615
C07951=1207.899,104.169,-49.517,-178.605,5.813,148.615
C07952=1207.904,103.919,-49.497,-178.607,5.812,148.616
C07953=1207.909,103.670,-49.478,-178.609,5.812,148.616
C07954=1207.914,103.421,-49.460,-178.612,5.810,148.617
C07955=1207.918,103.172,-49.441,-178.615,5.809,148.617
C07956=1207.924,102.922,-49.422,-178.617,5.808,148.618
C07957=1207.928,102.673,-49.403,-178.620,5.807,148.619
C07958=1207.933,102.424,-49.385,-178.623,5.806,148.619
C07959=1207.938,102.175,-49.366,-178.625,5.805,148.620
C07960=1207.943,101.925,-49.347,-178.628,5.804,148.620
C07961=1207.948,101.676,-49.328,-178.630,5.803,148.621
C07962=1207.953,101.427,-49.310,-178.633,5.802,148.621
C07963=1207.957,101.177,-49.292,-178.635,5.801,148.622
C07964=1207.962,100.928,-49.272,-178.638,5.800,148.622
C07965=1207.967,100.679,-49.254,-178.641,5.798,148.623
C07966=1207.971,100.430,-49.235,-178.643,5.798,148.623
C07967=1207.977,100.180,-49.217,-178.646,5.797,148.624
C07968=1207.982,99.932,-49.198,-178.649,5.795,148.624
C07969=1207.986,99.682,-49.180,-178.651,5.795,148.625
C07970=1207.992,99.432,-49.161,-178.653,5.794,148.626
C07971=1207.996,99.184,-49.143,-178.656,5.793,148.626
C07972=1208.001,98.934,-49.124,-178.659,5.792,148.627
C07973=1208.006,98.684,-49.106,-178.661,5.791,148.627
C07974=1208.011,98.436,-49.087,-178.664,5.789,148.628
C07975=1208.015,98.186,-49.069,-178.667,5.789,148.628
C07976=1208.020,97.937,-49.051,-178.669,5.788,148.629
C07977=1208.025,97.688,-49.031,-178.671,5.787,148.629
C07978=1208.030,97.439,-49.013,-178.674,5.786,148.630
C07979=1208.035,97.189,-48.995,-178.677,5.785,148.630
C07980=1208.040,96.940,-48.976,-178.679,5.784,148.631
C07981=1208.045,96.691,-48.958,-178.682,5.782,148.631
C07982=1208.049,96.441,-48.939,-178.685,5.782,148.632
C07983=1208.054,96.192,-48.921,-178.687,5.781,148.633
C07984=1208.059,95.943,-48.903,-178.690,5.780,148.633
C07985=1208.064,95.694,-48.884,-178.692,5.779,148.634
C07986=1208.069,95.444,-48.866,-178.695,5.778,148.634
C07987=1208.074,95.195,-48.848,-178.698,5.777,148.635
C07988=1208.078,94.946,-48.829,-178.700,5.776,148.636
C07989=1208.084,94.697,-48.811,-178.703,5.775,148.636
C07990=1208.088,94.447,-48.792,-178.705,5.775,148.637
C07991=1208.093,94.198,-48.774,-178.708,5.773,148.637
C07992=1208.098,93.948,-48.756,-178.710,5.772,148.638
C07993=1208.103,93.700,-48.738,-178.713,5.771,148.638
C07994=1208.107,93.450,-48.719,-178.716,5.770,148.639
C07995=1208.113,93.201,-48.701,-178.718,5.769,148.639
C07996=1208.117,92.951,-48.683,-178.721,5.768,148.640
C07997=1208.122,92.702,-48.665,-178.724,5.767,148.640
C07998=1208.127,92.453,-48.647,-178.726,5.766,148.641
C07999=1208.132,92.203,-48.628,-178.729,5.765,148.641
C08000=1208.136,91.954,-48.610,-178.731,5.765,148.642
C08001=1208.141,91.705,-48.592,-178.734,5.763,148.643
C08002=1208.147,91.456,-48.573,-178.736,5.763,148.643
C08003=1208.152,91.207,-48.555,-178.739,5.762,148.644
C08004=1208.156,90.957,-48.537,-178.741,5.761,148.644
C08005=1208.161,90.708,-48.519,-178.744,5.760,148.645
C08006=1208.166,90.458,-48.501,-178.747,5.759,148.645
C08007=1208.171,90.209,-48.483,-178.749,5.758,148.646
C08008=1208.176,89.960,-48.465,-178.752,5.756,148.646
C08009=1208.181,89.711,-48.447,-178.754,5.756,148.647
C08010=1208.185,89.461,-48.428,-178.757,5.755,148.648
C08011=1208.190,89.212,-48.410,-178.759,5.754,148.648
C08012=1208.195,88.963,-48.393,-178.762,5.753,148.649
C08013=1208.200,88.714,-48.375,-178.765,5.752,148.649
C08014=1208.204,88.464,-48.357,-178.767,5.751,148.650
C08015=1208.209,88.215,-48.339,-178.770,5.751,148.651
C08016=1208.214,87.966,-48.321,-178.773,5.749,148.651
C08017=1208.219,87.716,-48.302,-178.775,5.748,148.652
C08018=1208.224,87.467,-48.284,-178.778,5.748,148.652
C08019=1208.228,87.218,-48.266,-178.780,5.747,148.653
C08020=1208.233,86.969,-48.248,-178.783,5.746,148.653
C08021=1208.238,86.719,-48.230,-178.785,5.745,148.654
C08022=1208.243,86.470,-48.213,-178.788,5.744,148.654
C08023=1208.248,86.220,-48.195,-178.791,5.743,148.655
C08024=1208.253,85.971,-48.177,-178.793,5.742,148.655
C08025=1208.258,85.722,-48.159,-178.796,5.741,148.656
C08026=1208.263,85.473,-48.141,-178.798,5.741,148.657
C08027=1208.267,85.223,-48.123,-178.801,5.739,148.657
C08028=1208.272,84.974,-48.105,-178.804,5.738,148.658
C08029=1208.277,84.725,-48.087,-178.806,5.737,148.658
C08030=1208.282,84.475,-48.070,-178.809,5.737,148.659
C08031=1208.287,84.226,-48.052,-178.811,5.736,148.660
C08032=1208.292,83.977,-48.034,-178.814,5.734,148.660
C08033=1208.297,83.727,-48.016,-178.816,5.734,148.661
C08034=1208.302,83.478,-47.998,-178.819,5.733,148.661
C08035=1208.307,83.228,-47.980,-178.821,5.732,148.662
C08036=1208.312,82.979,-47.962,-178.824,5.731,148.662
C08037=1208.317,82.730,-47.944,-178.827,5.730,148.663
C08038=1208.321,82.481,-47.927,-178.829,5.729,148.663
C08039=1208.327,82.231,-47.910,-178.832,5.729,148.664
C08040=1208.331,81.982,-47.892,-178.835,5.727,148.664
C08041=1208.336,81.733,-47.874,-178.837,5.727,148.665
C08042=1208.342,81.464,-47.855,-178.840,5.726,148.666
C08043=1208.347,81.196,-47.836,-178.843,5.725,148.666
C08044=1208.352,80.928,-47.816,-178.846,5.724,148.667
C08045=1208.357,80.659,-47.798,-178.848,5.723,148.668
C08046=1208.362,80.410,-47.780,-178.851,5.722,148.668
C08047=1208.366,80.161,-47.762,-178.854,5.721,148.669
C08048=1208.372,79.911,-47.745,-178.856,5.720,148.669
C08049=1208.377,79.662,-47.727,-178.858,5.720,148.670
C08050=1208.381,79.413,-47.709,-178.861,5.719,148.671
C08051=1208.387,79.163,-47.692,-178.864,5.717,148.671
C08052=1208.392,78.914,-47.674,-178.866,5.717,148.672
C08053=1208.396,78.664,-47.657,-178.869,5.716,148.672
C08054=1208.401,78.415,-47.639,-178.871,5.715,148.673
C08055=1208.406,78.166,-47.621,-178.874,5.715,148.673
C08056=1208.411,77.916,-47.604,-178.877,5.713,148.674
C08057=1208.415,77.667,-47.587,-178.879,5.712,148.674
C08058=1208.420,77.417,-47.569,-178.882,5.712,148.675
C08059=1208.425,77.168,-47.551,-178.884,5.711,148.676
C08060=1208.430,76.919,-47.533,-178.887,5.710,148.676
C08061=1208.435,76.670,-47.517,-178.890,5.709,148.677
C08062=1208.440,76.421,-47.499,-178.892,5.708,148.678
C08063=1208.446,76.171,-47.482,-178.894,5.707,148.678
C08064=1208.450,75.922,-47.464,-178.897,5.707,148.679
C08065=1208.455,75.673,-47.447,-178.900,5.706,148.679
C08066=1208.460,75.423,-47.429,-178.902,5.705,148.680
C08067=1208.465,75.174,-47.412,-178.905,5.704,148.680
C08068=1208.469,74.925,-47.394,-178.908,5.703,148.681
C08069=1208.474,74.675,-47.377,-178.910,5.703,148.681
C08070=1208.479,74.426,-47.359,-178.912,5.702,148.682
C08071=1208.485,74.176,-47.342,-178.916,5.701,148.683
C08072=1208.489,73.927,-47.325,-178.918,5.700,148.683
C08073=1208.494,73.677,-47.307,-178.920,5.699,148.684
C08074=1208.500,73.428,-47.290,-178.923,5.699,148.684
C08075=1208.504,73.179,-47.273,-178.926,5.698,148.685
C08076=1208.509,72.930,-47.256,-178.928,5.696,148.686
C08077=1208.513,72.681,-47.238,-178.931,5.696,148.686
C08078=1208.519,72.431,-47.221,-178.934,5.695,148.687
C08079=1208.524,72.181,-47.204,-178.936,5.694,148.687
C08080=1208.528,71.932,-47.186,-178.938,5.694,148.688
C08081=1208.533,71.682,-47.169,-178.941,5.693,148.689
C08082=1208.539,71.434,-47.152,-178.944,5.691,148.689
C08083=1208.543,71.185,-47.135,-178.946,5.691,148.690
C08084=1208.548,70.935,-47.118,-178.949,5.690,148.690
C08085=1208.553,70.686,-47.100,-178.951,5.689,148.691
C08086=1208.558,70.436,-47.083,-178.954,5.689,148.691
C08087=1208.563,70.186,-47.066,-178.956,5.688,148.692
C08088=1208.567,69.937,-47.049,-178.959,5.686,148.693
C08089=1208.573,69.688,-47.031,-178.962,5.686,148.693
C08090=1208.577,69.439,-47.015,-178.964,5.685,148.694
C08091=1208.583,69.189,-46.998,-178.967,5.685,148.695
C08092=1208.587,68.940,-46.980,-178.969,5.684,148.695
C08093=1208.592,68.690,-46.963,-178.972,5.683,148.696
C08094=1208.597,68.441,-46.946,-178.974,5.683,148.696
C08095=1208.602,68.192,-46.929,-178.977,5.681,148.697
C08096=1208.607,67.943,-46.912,-178.980,5.680,148.697
C08097=1208.612,67.693,-46.895,-178.982,5.680,148.698
C08098=1208.616,67.444,-46.878,-178.984,5.679,148.698
C08099=1208.621,67.194,-46.861,-178.987,5.678,148.699
C08100=1208.627,66.945,-46.844,-178.990,5.678,148.700
C08101=1208.631,66.696,-46.826,-178.993,5.676,148.700
C08102=1208.636,66.446,-46.810,-178.995,5.675,148.701
C08103=1208.641,66.197,-46.792,-178.998,5.675,148.702
C08104=1208.646,65.947,-46.776,-179.000,5.674,148.702
C08105=1208.651,65.698,-46.759,-179.002,5.673,148.703
C08106=1208.656,65.449,-46.742,-179.005,5.673,148.703
C08107=1208.661,65.199,-46.724,-179.008,5.672,148.704
C08108=1208.665,64.950,-46.708,-179.010,5.672,148.705
C08109=1208.671,64.701,-46.691,-179.013,5.670,148.705
C08110=1208.676,64.451,-46.674,-179.016,5.670,148.706
C08111=1208.681,64.202,-46.657,-179.018,5.669,148.706
C08112=1208.685,63.952,-46.640,-179.020,5.668,148.707
C08113=1208.690,63.703,-46.624,-179.023,5.667,148.708
C08114=1208.696,63.453,-46.607,-179.026,5.667,148.708
C08115=1208.700,63.204,-46.590,-179.028,5.666,148.709
C08116=1208.705,62.954,-46.573,-179.031,5.665,148.709
C08117=1208.710,62.706,-46.556,-179.034,5.664,148.710
C08118=1208.715,62.457,-46.539,-179.036,5.664,148.711
C08119=1208.720,62.207,-46.522,-179.039,5.663,148.711
C08120=1208.725,61.958,-46.505,-179.041,5.662,148.712
C08121=1208.729,61.708,-46.489,-179.044,5.661,148.712
C08122=1208.735,61.459,-46.471,-179.046,5.661,148.713
C08123=1208.739,61.209,-46.455,-179.049,5.660,148.713
C08124=1208.745,60.960,-46.438,-179.051,5.659,148.714
C08125=1208.749,60.711,-46.421,-179.054,5.658,148.715
C08126=1208.754,60.461,-46.405,-179.057,5.658,148.715
C08127=1208.760,60.212,-46.388,-179.059,5.657,148.716
C08128=1208.764,59.962,-46.372,-179.062,5.656,148.717
C08129=1208.769,59.712,-46.355,-179.064,5.656,148.717
C08130=1208.775,59.463,-46.338,-179.067,5.655,148.718
C08131=1208.779,59.214,-46.321,-179.069,5.654,148.718
C08132=1208.784,58.964,-46.305,-179.072,5.654,148.719
C08133=1208.789,58.716,-46.288,-179.074,5.653,148.720
C08134=1208.794,58.466,-46.271,-179.078,5.652,148.720
C08135=1208.798,58.216,-46.255,-179.080,5.651,148.721
C08136=1208.804,57.968,-46.238,-179.082,5.650,148.721
C08137=1208.809,57.718,-46.221,-179.085,5.650,148.722
C08138=1208.813,57.468,-46.204,-179.087,5.649,148.723
C08139=1208.819,57.219,-46.189,-179.090,5.648,148.723
C08140=1208.823,56.969,-46.172,-179.092,5.648,148.724
C08141=1208.829,56.720,-46.155,-179.095,5.647,148.725
C08142=1208.833,56.471,-46.138,-179.097,5.646,148.725
C08143=1208.838,56.221,-46.122,-179.100,5.646,148.726
C08144=1208.843,55.973,-46.105,-179.103,5.645,148.726
C08145=1208.848,55.722,-46.089,-179.106,5.644,148.727
C08146=1208.854,55.454,-46.071,-179.108,5.643,148.728
C08147=1208.858,55.186,-46.053,-179.111,5.643,148.728
C08148=1208.864,54.917,-46.036,-179.114,5.642,148.729
C08149=1208.869,54.648,-46.017,-179.116,5.641,148.730
C08150=1208.875,54.399,-46.002,-179.119,5.640,148.730
C08151=1208.879,54.149,-45.985,-179.122,5.639,148.731
C08152=1208.884,53.901,-45.969,-179.124,5.639,148.731
C08153=1208.889,53.651,-45.952,-179.127,5.638,148.732
C08154=1208.895,53.401,-45.936,-179.129,5.637,148.732
C08155=1208.899,53.152,-45.919,-179.132,5.637,148.733
C08156=1208.904,52.902,-45.903,-179.134,5.636,148.734
C08157=1208.909,52.654,-45.886,-179.137,5.636,148.734
C08158=1208.914,52.404,-45.870,-179.139,5.635,148.735
C08159=1208.919,52.155,-45.854,-179.142,5.634,148.736
C08160=1208.923,51.905,-45.837,-179.144,5.634,148.736
C08161=1208.929,51.656,-45.821,-179.147,5.633,148.737
C08162=1208.934,51.406,-45.805,-179.149,5.632,148.737
C08163=1208.938,51.157,-45.788,-179.152,5.632,148.738
C08164=1208.944,50.907,-45.772,-179.155,5.630,148.739
C08165=1208.948,50.658,-45.756,-179.158,5.630,148.739
C08166=1208.954,50.408,-45.740,-179.160,5.629,148.740
C08167=1208.958,50.159,-45.723,-179.162,5.628,148.740
C08168=1208.963,49.910,-45.707,-179.165,5.628,148.741
C08169=1208.968,49.660,-45.691,-179.168,5.627,148.742
C08170=1208.973,49.411,-45.675,-179.170,5.627,148.742
C08171=1208.978,49.161,-45.659,-179.173,5.626,148.743
C08172=1208.984,48.912,-45.642,-179.175,5.625,148.744
C08173=1208.988,48.663,-45.625,-179.178,5.625,148.744
C08174=1208.994,48.413,-45.610,-179.180,5.624,148.745
C08175=1208.998,48.164,-45.593,-179.183,5.623,148.745
C08176=1209.003,47.914,-45.577,-179.185,5.623,148.746
C08177=1209.008,47.665,-45.561,-179.188,5.622,148.747
C08178=1209.013,47.415,-45.545,-179.190,5.621,148.747
C08179=1209.018,47.166,-45.529,-179.193,5.621,148.748
C08180=1209.023,46.916,-45.513,-179.195,5.620,148.749
C08181=1209.028,46.667,-45.496,-179.198,5.619,148.749
C08182=1209.033,46.418,-45.481,-179.201,5.619,148.750
C08183=1209.037,46.168,-45.464,-179.203,5.618,148.751
C08184=1209.043,45.919,-45.448,-179.206,5.617,148.751
C08185=1209.047,45.669,-45.432,-179.209,5.616,148.752
C08186=1209.053,45.420,-45.416,-179.211,5.616,148.752
C08187=1209.058,45.171,-45.400,-179.214,5.615,148.753
C08188=1209.063,44.921,-45.384,-179.216,5.614,148.754
C08189=1209.068,44.672,-45.368,-179.219,5.614,148.754
C08190=1209.072,44.422,-45.352,-179.221,5.613,148.755
C08191=1209.078,44.173,-45.336,-179.224,5.612,148.755
C08192=1209.082,43.923,-45.320,-179.227,5.612,148.756
C08193=1209.087,43.674,-45.304,-179.229,5.611,148.757
C08194=1209.092,43.425,-45.289,-179.231,5.611,148.757
C08195=1209.097,43.175,-45.272,-179.234,5.610,148.758
C08196=1209.102,42.926,-45.257,-179.237,5.609,148.759
C08197=1209.107,42.676,-45.241,-179.239,5.609,148.759
C08198=1209.112,42.427,-45.224,-179.241,5.608,148.760
C08199=1209.117,42.177,-45.209,-179.244,5.607,148.760
C08200=1209.122,41.927,-45.193,-179.247,5.607,148.761
C08201=1209.127,41.679,-45.176,-179.249,5.606,148.762
C08202=1209.132,41.428,-45.161,-179.252,5.606,148.762
C08203=1209.137,41.179,-45.146,-179.254,5.605,148.763
C08204=1209.142,40.931,-45.129,-179.257,5.604,148.763
C08205=1209.147,40.681,-45.113,-179.259,5.604,148.764
C08206=1209.152,40.431,-45.098,-179.262,5.603,148.765
C08207=1209.157,40.182,-45.081,-179.265,5.603,148.766
C08208=1209.162,39.932,-45.065,-179.267,5.602,148.766
C08209=1209.167,39.683,-45.050,-179.269,5.601,148.767
C08210=1209.171,39.433,-45.034,-179.272,5.601,148.767
C08211=1209.176,39.184,-45.018,-179.275,5.600,148.768
C08212=1209.182,38.935,-45.003,-179.277,5.600,148.769
C08213=1209.187,38.685,-44.987,-179.280,5.599,148.769
C08214=1209.192,38.435,-44.971,-179.282,5.598,148.770
C08215=1209.197,38.186,-44.955,-179.285,5.598,148.770
C08216=1209.201,37.937,-44.939,-179.287,5.597,148.771
C08217=1209.206,37.687,-44.924,-179.290,5.597,148.772
C08218=1209.212,37.438,-44.908,-179.293,5.596,148.772
C08219=1209.217,37.188,-44.892,-179.295,5.595,148.773
C08220=1209.222,36.938,-44.877,-179.298,5.595,148.774
C08221=1209.227,36.689,-44.862,-179.300,5.594,148.774
C08222=1209.231,36.440,-44.845,-179.303,5.594,148.775
C08223=1209.237,36.190,-44.829,-179.305,5.593,148.776
C08224=1209.242,35.941,-44.814,-179.308,5.592,148.776
C08225=1209.246,35.691,-44.798,-179.310,5.592,148.777
C08226=1209.251,35.442,-44.783,-179.313,5.591,148.777
C08227=1209.257,35.192,-44.767,-179.316,5.591,148.778
C08228=1209.262,34.943,-44.752,-179.318,5.590,148.779
C08229=1209.266,34.693,-44.736,-179.320,5.589,148.779
C08230=1209.272,34.444,-44.721,-179.323,5.589,148.780
C08231=1209.277,34.195,-44.704,-179.326,5.588,148.781
C08232=1209.281,33.945,-44.689,-179.328,5.588,148.781
C08233=1209.286,33.696,-44.673,-179.331,5.587,148.782
C08234=1209.292,33.447,-44.658,-179.334,5.587,148.783
C08235=1209.296,33.197,-44.643,-179.336,5.586,148.783
C08236=1209.301,32.947,-44.627,-179.338,5.585,148.784
C08237=1209.306,32.698,-44.611,-179.341,5.585,148.784
C08238=1209.311,32.449,-44.596,-179.344,5.584,148.785
C08239=1209.316,32.199,-44.581,-179.346,5.584,148.786
C08240=1209.321,31.949,-44.565,-179.348,5.583,148.786
C08241=1209.326,31.700,-44.550,-179.351,5.582,148.787
C08242=1209.331,31.451,-44.534,-179.353,5.582,148.788
C08243=1209.337,31.201,-44.519,-179.356,5.582,148.788
C08244=1209.341,30.952,-44.503,-179.358,5.581,148.789
C08245=1209.346,30.702,-44.488,-179.361,5.581,148.790
C08246=1209.351,30.453,-44.472,-179.363,5.580,148.790
C08247=1209.356,30.203,-44.458,-179.366,5.579,148.791
C08248=1209.362,29.954,-44.442,-179.369,5.579,148.791
C08249=1209.366,29.704,-44.427,-179.371,5.578,148.792
C08250=1209.371,29.435,-44.410,-179.374,5.578,148.793
C08251=1209.377,29.166,-44.394,-179.376,5.577,148.793
C08252=1209.382,28.898,-44.377,-179.380,5.576,148.794
C08253=1209.388,28.630,-44.360,-179.382,5.575,148.795
C08254=1209.393,28.380,-44.345,-179.385,5.575,148.795
C08255=1209.398,28.131,-44.330,-179.388,5.574,148.796
C08256=1209.403,27.881,-44.315,-179.390,5.575,148.797
C08257=1209.407,27.631,-44.299,-179.392,5.574,148.797
C08258=1209.413,27.382,-44.284,-179.394,5.573,148.798
C08259=1209.417,27.133,-44.269,-179.397,5.573,148.799
C08260=1209.423,26.883,-44.253,-179.400,5.572,148.799
C08261=1209.428,26.634,-44.239,-179.402,5.572,148.800
C08262=1209.433,26.384,-44.223,-179.405,5.571,148.801
C08263=1209.438,26.134,-44.207,-179.407,5.570,148.801
C08264=1209.443,25.885,-44.192,-179.410,5.570,148.802
C08265=1209.448,25.636,-44.177,-179.412,5.569,148.802
C08266=1209.453,25.386,-44.162,-179.415,5.569,148.803
C08267=1209.458,25.137,-44.147,-179.418,5.568,148.804
C08268=1209.463,24.888,-44.132,-179.420,5.568,148.804
C08269=1209.468,24.637,-44.116,-179.423,5.567,148.805
C08270=1209.473,24.388,-44.102,-179.425,5.566,148.806
C08271=1209.477,24.139,-44.087,-179.428,5.566,148.806
C08272=1209.483,23.889,-44.071,-179.430,5.566,148.807
C08273=1209.487,23.640,-44.056,-179.433,5.565,148.808
C08274=1209.493,23.390,-44.041,-179.435,5.565,148.808
C08275=1209.498,23.141,-44.026,-179.438,5.564,148.809
C08276=1209.503,22.892,-44.011,-179.440,5.563,148.809
C08277=1209.508,22.642,-43.996,-179.443,5.563,148.810
C08278=1209.513,22.392,-43.980,-179.445,5.562,148.811
C08279=1209.517,22.143,-43.965,-179.448,5.562,148.812
C08280=1209.522,21.893,-43.951,-179.451,5.561,148.812
C08281=1209.528,21.644,-43.936,-179.453,5.561,148.813
C08282=1209.532,21.395,-43.921,-179.456,5.560,148.814
C08283=1209.538,21.145,-43.906,-179.458,5.559,148.814
C08284=1209.543,20.895,-43.891,-179.461,5.559,148.815
C08285=1209.549,20.645,-43.876,-179.463,5.559,148.815
C08286=1209.553,20.396,-43.861,-179.465,5.559,148.816
C08287=1209.558,20.147,-43.846,-179.468,5.558,148.817
C08288=1209.563,19.897,-43.831,-179.471,5.558,148.817
C08289=1209.568,19.648,-43.816,-179.473,5.557,148.818
C08290=1209.573,19.398,-43.802,-179.476,5.556,148.819
C08291=1209.578,19.149,-43.786,-179.478,5.556,148.819
C08292=1209.583,18.899,-43.771,-179.481,5.555,148.820
C08293=1209.587,18.649,-43.756,-179.483,5.555,148.821
C08294=1209.593,18.400,-43.741,-179.486,5.554,148.821
C08295=1209.598,18.150,-43.727,-179.489,5.554,148.822
C08296=1209.602,17.901,-43.712,-179.490,5.554,148.822
C08297=1209.608,17.651,-43.697,-179.493,5.553,148.823
C08298=1209.613,17.402,-43.682,-179.496,5.553,148.824
C08299=1209.618,17.152,-43.667,-179.498,5.552,148.824
C08300=1209.623,16.903,-43.652,-179.501,5.552,148.825
C08301=1209.628,16.653,-43.638,-179.504,5.551,148.826
C08302=1209.633,16.404,-43.623,-179.506,5.550,148.827
C08303=1209.638,16.154,-43.608,-179.508,5.550,148.827
C08304=1209.643,15.905,-43.593,-179.511,5.549,148.828
C08305=1209.648,15.655,-43.578,-179.514,5.549,148.828
C08306=1209.653,15.406,-43.563,-179.516,5.549,148.829
C08307=1209.658,15.156,-43.549,-179.518,5.548,148.830
C08308=1209.663,14.907,-43.534,-179.521,5.548,148.830
C08309=1209.668,14.658,-43.519,-179.524,5.547,148.831
C08310=1209.674,14.407,-43.504,-179.526,5.547,148.832
C08311=1209.678,14.158,-43.489,-179.529,5.546,148.832
C08312=1209.683,13.909,-43.475,-179.531,5.545,148.833
C08313=1209.688,13.660,-43.460,-179.534,5.545,148.834
C08314=1209.693,13.410,-43.446,-179.536,5.545,148.834
C08315=1209.699,13.160,-43.431,-179.539,5.545,148.835
C08316=1209.704,12.911,-43.416,-179.541,5.544,148.836
C08317=1209.709,12.662,-43.402,-179.544,5.544,148.836
C08318=1209.714,12.412,-43.388,-179.546,5.543,148.837
C08319=1209.719,12.163,-43.372,-179.549,5.542,148.837
C08320=1209.724,11.913,-43.358,-179.551,5.542,148.838
C08321=1209.729,11.663,-43.344,-179.554,5.541,148.839
C08322=1209.734,11.414,-43.329,-179.557,5.541,148.839
C08323=1209.739,11.164,-43.314,-179.559,5.541,148.840
C08324=1209.744,10.915,-43.300,-179.561,5.540,148.841
C08325=1209.749,10.665,-43.285,-179.564,5.540,148.842
C08326=1209.754,10.416,-43.270,-179.566,5.539,148.842
C08327=1209.759,10.166,-43.256,-179.569,5.539,148.843
C08328=1209.764,9.916,-43.242,-179.571,5.538,148.843
C08329=1209.769,9.667,-43.227,-179.574,5.538,148.844
C08330=1209.774,9.418,-43.213,-179.576,5.538,148.845
C08331=1209.779,9.168,-43.199,-179.579,5.537,148.845
C08332=1209.785,8.918,-43.184,-179.581,5.537,148.846
C08333=1209.789,8.669,-43.169,-179.584,5.536,148.847
C08334=1209.794,8.420,-43.154,-179.586,5.535,148.847
C08335=1209.799,8.170,-43.140,-179.589,5.535,148.848
C08336=1209.804,7.920,-43.126,-179.592,5.534,148.849
C08337=1209.809,7.671,-43.111,-179.594,5.535,148.849
C08338=1209.814,7.421,-43.097,-179.596,5.534,148.850
C08339=1209.819,7.172,-43.083,-179.599,5.534,148.851
C08340=1209.824,6.923,-43.068,-179.602,5.533,148.851
C08341=1209.829,6.673,-43.054,-179.604,5.533,148.852
C08342=1209.835,6.423,-43.039,-179.606,5.532,148.853
C08343=1209.840,6.174,-43.024,-179.609,5.531,148.853
C08344=1209.845,5.924,-43.010,-179.611,5.532,148.854
C08345=1209.850,5.674,-42.996,-179.614,5.531,148.855
C08346=1209.855,5.425,-42.982,-179.616,5.531,148.855
C08347=1209.860,5.176,-42.968,-179.619,5.530,148.856
C08348=1209.865,4.926,-42.953,-179.622,5.530,148.857
C08349=1209.870,4.676,-42.939,-179.624,5.529,148.857
C08350=1209.875,4.427,-42.925,-179.627,5.528,148.858
C08351=1209.880,4.177,-42.910,-179.629,5.528,148.858
C08352=1209.885,3.928,-42.896,-179.631,5.528,148.859
C08353=1209.890,3.679,-42.882,-179.634,5.527,148.860
C08354=1209.896,3.409,-42.867,-179.637,5.527,148.861
C08355=1209.901,3.141,-42.851,-179.639,5.526,148.861
C08356=1209.906,2.871,-42.836,-179.642,5.526,148.862
C08357=1209.911,2.602,-42.820,-179.645,5.526,148.863
C08358=1209.917,2.353,-42.806,-179.647,5.525,148.863
C08359=1209.922,2.104,-42.792,-179.650,5.524,148.864
C08360=1209.927,1.854,-42.778,-179.652,5.525,148.865
C08361=1209.932,1.604,-42.763,-179.655,5.524,148.865
C08362=1209.937,1.354,-42.749,-179.657,5.524,148.866
C08363=1209.942,1.105,-42.735,-179.660,5.523,148.867
C08364=1209.947,0.856,-42.721,-179.663,5.523,148.867
C08365=1209.952,0.606,-42.707,-179.665,5.522,148.868
C08366=1209.957,0.356,-42.692,-179.667,5.523,148.869
C08367=1209.963,0.107,-42.678,-179.669,5.522,148.869
C08368=1209.968,-0.143,-42.665,-179.672,5.521,148.870
C08369=1209.973,-0.393,-42.651,-179.675,5.521,148.871
C08370=1209.978,-0.642,-42.636,-179.677,5.520,148.871
C08371=1209.983,-0.891,-42.622,-179.680,5.520,148.872
C08372=1209.987,-1.141,-42.609,-179.682,5.520,148.873
C08373=1209.992,-1.391,-42.594,-179.685,5.519,148.873
C08374=1209.997,-1.640,-42.580,-179.687,5.519,148.874
C08375=1210.003,-1.889,-42.566,-179.690,5.518,148.875
C08376=1210.008,-2.139,-42.552,-179.692,5.518,148.875
C08377=1210.013,-2.389,-42.538,-179.694,5.518,148.876
C08378=1210.018,-2.638,-42.523,-179.697,5.517,148.877
C08379=1210.024,-2.888,-42.510,-179.700,5.517,148.877
C08380=1210.028,-3.137,-42.497,-179.702,5.516,148.878
C08381=1210.033,-3.387,-42.482,-179.705,5.516,148.879
C08382=1210.038,-3.636,-42.468,-179.707,5.516,148.879
C08383=1210.043,-3.886,-42.454,-179.710,5.516,148.880
C08384=1210.048,-4.136,-42.440,-179.712,5.515,148.881
C08385=1210.054,-4.386,-42.426,-179.715,5.515,148.881
C08386=1210.058,-4.635,-42.413,-179.717,5.514,148.882
C08387=1210.063,-4.884,-42.399,-179.720,5.513,148.883
C08388=1210.068,-5.134,-42.384,-179.722,5.514,148.883
C08389=1210.074,-5.383,-42.370,-179.725,5.513,148.884
C08390=1210.079,-5.633,-42.357,-179.727,5.513,148.885
C08391=1210.083,-5.883,-42.343,-179.730,5.512,148.885
C08392=1210.089,-6.132,-42.329,-179.732,5.512,148.886
C08393=1210.094,-6.381,-42.315,-179.735,5.512,148.887
C08394=1210.099,-6.632,-42.302,-179.737,5.511,148.887
C08395=1210.105,-6.881,-42.288,-179.739,5.511,148.888
C08396=1210.109,-7.130,-42.274,-179.742,5.510,148.889
C08397=1210.114,-7.380,-42.260,-179.744,5.510,148.889
C08398=1210.120,-7.630,-42.246,-179.747,5.510,148.890
C08399=1210.125,-7.879,-42.232,-179.749,5.509,148.891
C08400=1210.129,-8.129,-42.218,-179.752,5.509,148.891
C08401=1210.135,-8.378,-42.205,-179.755,5.508,148.892
C08402=1210.140,-8.628,-42.191,-179.757,5.509,148.893
C08403=1210.144,-8.877,-42.177,-179.759,5.508,148.893
C08404=1210.150,-9.127,-42.164,-179.762,5.508,148.894
C08405=1210.155,-9.377,-42.150,-179.764,5.507,148.895
C08406=1210.160,-9.626,-42.136,-179.767,5.506,148.895
C08407=1210.165,-9.876,-42.123,-179.769,5.507,148.896
C08408=1210.170,-10.126,-42.109,-179.772,5.506,148.897
C08409=1210.175,-10.375,-42.095,-179.774,5.506,148.897
C08410=1210.180,-10.625,-42.082,-179.777,5.505,148.898
C08411=1210.185,-10.874,-42.068,-179.779,5.506,148.899
C08412=1210.191,-11.124,-42.054,-179.782,5.505,148.899
C08413=1210.195,-11.373,-42.041,-179.784,5.505,148.900
C08414=1210.200,-11.622,-42.027,-179.787,5.504,148.901
C08415=1210.206,-11.873,-42.013,-179.789,5.503,148.901
C08416=1210.210,-12.122,-42.000,-179.791,5.503,148.902
C08417=1210.216,-12.372,-41.986,-179.794,5.503,148.903
C08418=1210.221,-12.621,-41.972,-179.797,5.503,148.903
C08419=1210.226,-12.871,-41.959,-179.799,5.502,148.904
C08420=1210.231,-13.120,-41.945,-179.801,5.502,148.905
C08421=1210.236,-13.369,-41.931,-179.804,5.502,148.905
C08422=1210.241,-13.619,-41.918,-179.807,5.501,148.906
C08423=1210.246,-13.869,-41.904,-179.809,5.501,148.907
C08424=1210.251,-14.118,-41.891,-179.812,5.500,148.907
C08425=1210.256,-14.368,-41.877,-179.814,5.500,148.908
C08426=1210.262,-14.618,-41.864,-179.816,5.500,148.909
C08427=1210.266,-14.867,-41.850,-179.819,5.499,148.909
C08428=1210.272,-15.117,-41.837,-179.822,5.499,148.910
C08429=1210.276,-15.366,-41.823,-179.824,5.499,148.911
C08430=1210.282,-15.616,-41.810,-179.826,5.499,148.911
C08431=1210.287,-15.866,-41.797,-179.829,5.498,148.912
C08432=1210.292,-16.115,-41.783,-179.832,5.498,148.913
C08433=1210.297,-16.365,-41.770,-179.834,5.498,148.914
C08434=1210.302,-16.614,-41.756,-179.836,5.498,148.914
C08435=1210.307,-16.864,-41.743,-179.839,5.497,148.915
C08436=1210.312,-17.113,-41.730,-179.841,5.496,148.915
C08437=1210.317,-17.363,-41.716,-179.843,5.496,148.916
C08438=1210.323,-17.613,-41.703,-179.846,5.496,148.917
C08439=1210.328,-17.862,-41.689,-179.849,5.495,148.917
C08440=1210.333,-18.112,-41.676,-179.851,5.495,148.918
C08441=1210.338,-18.361,-41.662,-179.853,5.495,148.919
C08442=1210.343,-18.611,-41.649,-179.856,5.495,148.920
C08443=1210.348,-18.861,-41.636,-179.859,5.494,148.920
C08444=1210.354,-19.110,-41.622,-179.861,5.494,148.921
C08445=1210.358,-19.360,-41.609,-179.863,5.494,148.922
C08446=1210.364,-19.610,-41.596,-179.866,5.494,148.922
C08447=1210.368,-19.859,-41.582,-179.868,5.493,148.923
C08448=1210.374,-20.109,-41.569,-179.871,5.492,148.923
C08449=1210.379,-20.359,-41.556,-179.873,5.493,148.924
C08450=1210.383,-20.607,-41.543,-179.876,5.492,148.925
C08451=1210.389,-20.858,-41.529,-179.878,5.492,148.926
C08452=1210.394,-21.107,-41.517,-179.881,5.491,148.926
C08453=1210.399,-21.357,-41.502,-179.883,5.492,148.927
C08454=1210.404,-21.606,-41.490,-179.886,5.491,148.928
C08455=1210.410,-21.856,-41.477,-179.888,5.491,148.928
C08456=1210.414,-22.106,-41.464,-179.891,5.490,148.929
C08457=1210.420,-22.355,-41.450,-179.893,5.490,148.930
C08458=1210.425,-22.624,-41.436,-179.896,5.490,148.930
C08459=1210.430,-22.894,-41.422,-179.898,5.489,148.931
C08460=1210.436,-23.163,-41.408,-179.901,5.489,148.932
C08461=1210.442,-23.433,-41.393,-179.904,5.488,148.933
C08462=1210.446,-23.683,-41.380,-179.906,5.488,148.933
C08463=1210.452,-23.932,-41.367,-179.908,5.488,148.934
C08464=1210.457,-24.181,-41.354,-179.911,5.488,148.935
C08465=1210.462,-24.432,-41.340,-179.914,5.487,148.935
C08466=1210.467,-24.681,-41.328,-179.916,5.488,148.936
C08467=1210.472,-24.931,-41.315,-179.918,5.487,148.937
C08468=1210.477,-25.180,-41.301,-179.921,5.486,148.937
C08469=1210.482,-25.429,-41.288,-179.923,5.486,148.938
C08470=1210.487,-25.679,-41.275,-179.925,5.486,148.939
C08471=1210.493,-25.929,-41.262,-179.928,5.486,148.939
C08472=1210.497,-26.179,-41.249,-179.931,5.485,148.940
C08473=1210.502,-26.428,-41.237,-179.933,5.486,148.941
C08474=1210.508,-26.677,-41.223,-179.935,5.485,148.941
C08475=1210.512,-26.927,-41.210,-179.938,5.485,148.942
C08476=1210.518,-27.177,-41.197,-179.941,5.484,148.943
C08477=1210.523,-27.426,-41.184,-179.943,5.484,148.943
C08478=1210.528,-27.676,-41.171,-179.945,5.484,148.944
C08479=1210.533,-27.926,-41.158,-179.948,5.483,148.945
C08480=1210.538,-28.176,-41.145,-179.950,5.483,148.945
C08481=1210.543,-28.425,-41.132,-179.952,5.483,148.946
C08482=1210.549,-28.674,-41.120,-179.955,5.482,148.947
C08483=1210.554,-28.925,-41.106,-179.958,5.482,148.947
C08484=1210.559,-29.174,-41.093,-179.960,5.482,148.948
C08485=1210.564,-29.423,-41.081,-179.962,5.482,148.949
C08486=1210.569,-29.673,-41.068,-179.965,5.481,148.949
C08487=1210.574,-29.923,-41.055,-179.967,5.482,148.950
C08488=1210.580,-30.172,-41.042,-179.970,5.481,148.951
C08489=1210.584,-30.422,-41.028,-179.972,5.481,148.952
C08490=1210.589,-30.671,-41.016,-179.975,5.480,148.952
C08491=1210.595,-30.921,-41.003,-179.977,5.480,148.953
C08492=1210.599,-31.171,-40.990,-179.979,5.480,148.953
C08493=1210.605,-31.421,-40.978,-179.982,5.479,148.954
C08494=1210.610,-31.670,-40.965,-179.984,5.480,148.955
C08495=1210.616,-31.920,-40.952,-179.987,5.479,148.956
C08496=1210.620,-32.170,-40.939,-179.989,5.479,148.956
C08497=1210.625,-32.419,-40.926,-179.992,5.479,148.957
C08498=1210.630,-32.668,-40.914,-179.994,5.478,148.958
C08499=1210.635,-32.918,-40.901,-179.997,5.478,148.958
C08500=1210.641,-33.168,-40.888,-180.000,5.478,148.959
C08501=1210.646,-33.417,-40.875,179.999,5.477,148.959
C08502=1210.651,-33.667,-40.862,179.996,5.477,148.960
C08503=1210.656,-33.917,-40.849,179.994,5.477,148.961
C08504=1210.661,-34.166,-40.837,179.991,5.477,148.962
C08505=1210.667,-34.416,-40.824,179.989,5.476,148.962
C08506=1210.671,-34.666,-40.811,179.986,5.476,148.963
C08507=1210.677,-34.916,-40.799,179.984,5.476,148.964
C08508=1210.682,-35.165,-40.786,179.981,5.476,148.964
C08509=1210.687,-35.414,-40.774,179.979,5.475,148.965
C08510=1210.691,-35.664,-40.761,179.977,5.476,148.966
C08511=1210.697,-35.914,-40.747,179.974,5.475,148.966
C08512=1210.702,-36.163,-40.735,179.971,5.475,148.967
C08513=1210.707,-36.412,-40.722,179.969,5.474,148.968
C08514=1210.713,-36.662,-40.710,179.967,5.474,148.968
C08515=1210.717,-36.912,-40.697,179.964,5.474,148.969
C08516=1210.723,-37.162,-40.685,179.962,5.473,148.970
C08517=1210.728,-37.411,-40.672,179.960,5.474,148.970
C08518=1210.733,-37.660,-40.660,179.957,5.473,148.971
C08519=1210.738,-37.911,-40.647,179.954,5.473,148.972
C08520=1210.743,-38.161,-40.634,179.952,5.473,148.973
C08521=1210.749,-38.410,-40.622,179.950,5.472,148.973
C08522=1210.754,-38.659,-40.609,179.947,5.472,148.974
C08523=1210.759,-38.909,-40.597,179.945,5.472,148.975
C08524=1210.764,-39.159,-40.584,179.943,5.471,148.975
C08525=1210.769,-39.409,-40.571,179.940,5.471,148.976
C08526=1210.774,-39.658,-40.559,179.938,5.471,148.977
C08527=1210.779,-39.908,-40.547,179.935,5.471,148.977
C08528=1210.784,-40.157,-40.534,179.933,5.470,148.978
C08529=1210.790,-40.406,-40.522,179.931,5.471,148.979
C08530=1210.794,-40.656,-40.509,179.928,5.470,148.979
C08531=1210.800,-40.906,-40.497,179.925,5.470,148.980
C08532=1210.805,-41.156,-40.484,179.923,5.470,148.981
C08533=1210.810,-41.405,-40.472,179.920,5.470,148.981
C08534=1210.815,-41.655,-40.460,179.918,5.469,148.982
C08535=1210.820,-41.905,-40.447,179.916,5.469,148.983
C08536=1210.825,-42.154,-40.434,179.914,5.469,148.983
C08537=1210.830,-42.404,-40.422,179.911,5.468,148.984
C08538=1210.835,-42.654,-40.410,179.909,5.469,148.985
C08539=1210.841,-42.903,-40.397,179.906,5.468,148.985
C08540=1210.846,-43.153,-40.385,179.903,5.468,148.986
C08541=1210.851,-43.402,-40.373,179.901,5.468,148.987
C08542=1210.856,-43.653,-40.360,179.899,5.467,148.987
C08543=1210.861,-43.902,-40.348,179.896,5.467,148.988
C08544=1210.866,-44.151,-40.335,179.894,5.467,148.989
C08545=1210.872,-44.401,-40.323,179.892,5.467,148.989
C08546=1210.877,-44.651,-40.311,179.889,5.466,148.990
C08547=1210.882,-44.901,-40.299,179.887,5.466,148.991
C08548=1210.887,-45.150,-40.286,179.884,5.466,148.991
C08549=1210.892,-45.399,-40.274,179.882,5.465,148.992
C08550=1210.898,-45.649,-40.262,179.880,5.466,148.993
C08551=1210.902,-45.899,-40.249,179.877,5.465,148.994
C08552=1210.908,-46.149,-40.237,179.874,5.465,148.994
C08553=1210.913,-46.398,-40.224,179.872,5.465,148.995
C08554=1210.918,-46.648,-40.212,179.870,5.465,148.996
C08555=1210.923,-46.898,-40.200,179.867,5.465,148.996
C08556=1210.928,-47.147,-40.189,179.865,5.464,148.997
C08557=1210.933,-47.397,-40.176,179.863,5.464,148.998
C08558=1210.939,-47.647,-40.164,179.861,5.464,148.998
C08559=1210.944,-47.896,-40.151,179.858,5.464,148.999
C08560=1210.949,-48.146,-40.140,179.855,5.463,149.000
C08561=1210.954,-48.395,-40.127,179.853,5.464,149.000
C08562=1210.960,-48.665,-40.114,179.850,5.463,149.001
C08563=1210.965,-48.936,-40.101,179.848,5.463,149.002
C08564=1210.971,-49.205,-40.088,179.845,5.462,149.002
C08565=1210.977,-49.476,-40.074,179.843,5.463,149.003
C08566=1210.981,-49.725,-40.063,179.840,5.462,149.004
C08567=1210.986,-49.974,-40.050,179.838,5.462,149.005
C08568=1210.992,-50.224,-40.038,179.836,5.462,149.005
C08569=1210.997,-50.474,-40.026,179.833,5.461,149.006
C08570=1211.002,-50.724,-40.014,179.830,5.461,149.007
C08571=1211.008,-50.974,-40.002,179.828,5.461,149.007
C08572=1211.012,-51.223,-39.990,179.826,5.461,149.008
C08573=1211.018,-51.473,-39.978,179.823,5.460,149.009
C08574=1211.023,-51.722,-39.966,179.821,5.461,149.010
C08575=1211.028,-51.972,-39.954,179.818,5.460,149.010
C08576=1211.034,-52.222,-39.942,179.817,5.460,149.011
C08577=1211.038,-52.471,-39.930,179.814,5.460,149.011
C08578=1211.043,-52.721,-39.918,179.811,5.459,149.012
C08579=1211.049,-52.971,-39.906,179.809,5.460,149.013
C08580=1211.054,-53.220,-39.893,179.806,5.459,149.014
C08581=1211.059,-53.470,-39.882,179.804,5.459,149.014
C08582=1211.064,-53.719,-39.870,179.802,5.459,149.015
C08583=1211.069,-53.969,-39.858,179.799,5.459,149.016
C08584=1211.075,-54.219,-39.846,179.797,5.459,149.016
C08585=1211.080,-54.469,-39.834,179.794,5.459,149.017
C08586=1211.085,-54.718,-39.822,179.792,5.458,149.018
C08587=1211.090,-54.968,-39.810,179.790,5.458,149.018
C08588=1211.095,-55.218,-39.798,179.787,5.458,149.019
C08589=1211.100,-55.467,-39.786,179.785,5.457,149.020
C08590=1211.105,-55.716,-39.774,179.783,5.457,149.020
C08591=1211.111,-55.966,-39.762,179.780,5.457,149.021
C08592=1211.116,-56.216,-39.750,179.778,5.457,149.022
C08593=1211.120,-56.465,-39.738,179.775,5.457,149.022
C08594=1211.126,-56.715,-39.727,179.773,5.456,149.023
C08595=1211.131,-56.965,-39.715,179.770,5.457,149.024
C08596=1211.136,-57.215,-39.703,179.768,5.456,149.024
C08597=1211.141,-57.464,-39.691,179.766,5.456,149.025
C08598=1211.147,-57.714,-39.679,179.764,5.456,149.026
C08599=1211.151,-57.964,-39.668,179.761,5.455,149.026
C08600=1211.157,-58.214,-39.656,179.759,5.456,149.027
C08601=1211.162,-58.464,-39.644,179.756,5.455,149.028
C08602=1211.167,-58.713,-39.633,179.753,5.455,149.029
C08603=1211.172,-58.963,-39.620,179.751,5.455,149.029
C08604=1211.177,-59.212,-39.608,179.749,5.455,149.030
C08605=1211.183,-59.461,-39.597,179.747,5.455,149.030
C08606=1211.188,-59.711,-39.585,179.744,5.454,149.031
C08607=1211.194,-59.961,-39.573,179.742,5.454,149.032
C08608=1211.198,-60.211,-39.562,179.740,5.454,149.033
C08609=1211.203,-60.460,-39.549,179.737,5.454,149.033
C08610=1211.208,-60.710,-39.538,179.735,5.454,149.034
C08611=1211.213,-60.960,-39.526,179.732,5.454,149.035
C08612=1211.219,-61.210,-39.514,179.730,5.453,149.035
C08613=1211.224,-61.459,-39.503,179.727,5.454,149.036
C08614=1211.229,-61.709,-39.491,179.725,5.453,149.037
C08615=1211.234,-61.958,-39.480,179.723,5.453,149.037
C08616=1211.240,-62.208,-39.468,179.721,5.453,149.038
C08617=1211.245,-62.458,-39.457,179.718,5.452,149.039
C08618=1211.250,-62.708,-39.445,179.716,5.452,149.039
C08619=1211.255,-62.958,-39.433,179.713,5.452,149.040
C08620=1211.260,-63.207,-39.421,179.711,5.452,149.041
C08621=1211.265,-63.457,-39.409,179.708,5.452,149.041
C08622=1211.270,-63.706,-39.398,179.706,5.451,149.042
C08623=1211.276,-63.955,-39.387,179.704,5.452,149.043
C08624=1211.280,-64.205,-39.375,179.701,5.451,149.043
C08625=1211.286,-64.455,-39.363,179.699,5.451,149.044
C08626=1211.291,-64.705,-39.352,179.697,5.451,149.045
C08627=1211.296,-64.955,-39.340,179.694,5.450,149.045
C08628=1211.301,-65.205,-39.328,179.692,5.451,149.046
C08629=1211.307,-65.453,-39.317,179.689,5.450,149.047
C08630=1211.312,-65.703,-39.306,179.687,5.451,149.048
C08631=1211.317,-65.953,-39.294,179.685,5.450,149.048
C08632=1211.322,-66.203,-39.282,179.682,5.449,149.049
C08633=1211.327,-66.453,-39.271,179.680,5.450,149.050
C08634=1211.333,-66.703,-39.260,179.678,5.449,149.050
C08635=1211.338,-66.952,-39.249,179.676,5.450,149.051
C08636=1211.343,-67.202,-39.237,179.673,5.449,149.052
C08637=1211.348,-67.452,-39.226,179.670,5.449,149.052
C08638=1211.354,-67.702,-39.214,179.668,5.449,149.053
C08639=1211.358,-67.951,-39.203,179.665,5.449,149.054
C08640=1211.364,-68.200,-39.191,179.663,5.449,149.054
C08641=1211.369,-68.450,-39.180,179.661,5.448,149.055
C08642=1211.374,-68.700,-39.168,179.659,5.449,149.056
C08643=1211.379,-68.950,-39.157,179.656,5.448,149.056
C08644=1211.384,-69.199,-39.145,179.654,5.448,149.057
C08645=1211.390,-69.449,-39.135,179.652,5.448,149.058
C08646=1211.395,-69.699,-39.123,179.649,5.448,149.058
C08647=1211.400,-69.949,-39.111,179.647,5.448,149.059
C08648=1211.405,-70.198,-39.100,179.644,5.448,149.060
C08649=1211.411,-70.447,-39.089,179.642,5.447,149.060
C08650=1211.416,-70.697,-39.077,179.640,5.447,149.061
C08651=1211.420,-70.947,-39.066,179.637,5.447,149.062
C08652=1211.426,-71.197,-39.055,179.635,5.447,149.062
C08653=1211.431,-71.446,-39.044,179.633,5.447,149.063
C08654=1211.437,-71.696,-39.032,179.630,5.447,149.064
C08655=1211.442,-71.946,-39.021,179.628,5.446,149.065
C08656=1211.446,-72.195,-39.009,179.625,5.446,149.065
C08657=1211.453,-72.445,-38.999,179.623,5.446,149.066
C08658=1211.457,-72.695,-38.987,179.621,5.446,149.066
C08659=1211.463,-72.945,-38.976,179.619,5.446,149.067
C08660=1211.467,-73.194,-38.964,179.616,5.445,149.068
C08661=1211.473,-73.444,-38.954,179.614,5.446,149.069
C08662=1211.478,-73.694,-38.942,179.611,5.445,149.069
C08663=1211.483,-73.944,-38.931,179.609,5.445,149.070
C08664=1211.488,-74.192,-38.920,179.607,5.445,149.071
C08665=1211.494,-74.443,-38.909,179.604,5.444,149.071
C08666=1211.499,-74.713,-38.896,179.602,5.445,149.072
C08667=1211.505,-74.983,-38.884,179.599,5.445,149.073
C08668=1211.511,-75.254,-38.872,179.596,5.444,149.074
C08669=1211.516,-75.525,-38.860,179.594,5.445,149.074
C08670=1211.521,-75.774,-38.849,179.592,5.444,149.075
C08671=1211.527,-76.025,-38.838,179.589,5.444,149.076
C08672=1211.532,-76.274,-38.827,179.587,5.444,149.076
C08673=1211.537,-76.523,-38.816,179.585,5.443,149.077
C08674=1211.543,-76.774,-38.805,179.583,5.444,149.078
C08675=1211.548,-77.024,-38.793,179.580,5.443,149.078
C08676=1211.553,-77.272,-38.782,179.578,5.444,149.079
C08677=1211.558,-77.523,-38.772,179.575,5.443,149.080
C08678=1211.563,-77.773,-38.760,179.573,5.444,149.080
C08679=1211.569,-78.022,-38.749,179.571,5.443,149.081
C08680=1211.574,-78.272,-38.738,179.568,5.442,149.082
C08681=1211.579,-78.522,-38.726,179.566,5.443,149.082
C08682=1211.585,-78.771,-38.716,179.564,5.442,149.083
C08683=1211.589,-79.021,-38.705,179.561,5.443,149.084
C08684=1211.594,-79.271,-38.694,179.559,5.442,149.084
C08685=1211.600,-79.520,-38.683,179.557,5.442,149.085
C08686=1211.605,-79.770,-38.672,179.555,5.442,149.086
C08687=1211.610,-80.020,-38.661,179.552,5.442,149.086
C08688=1211.615,-80.269,-38.650,179.550,5.442,149.087
C08689=1211.620,-80.519,-38.639,179.547,5.441,149.088
C08690=1211.626,-80.769,-38.628,179.545,5.441,149.088
C08691=1211.631,-81.018,-38.617,179.542,5.441,149.089
C08692=1211.636,-81.269,-38.606,179.540,5.441,149.090
C08693=1211.641,-81.517,-38.595,179.538,5.441,149.090
C08694=1211.646,-81.768,-38.585,179.536,5.441,149.091
C08695=1211.652,-82.017,-38.573,179.533,5.441,149.092
C08696=1211.657,-82.267,-38.563,179.531,5.441,149.093
C08697=1211.662,-82.517,-38.551,179.529,5.440,149.093
C08698=1211.668,-82.766,-38.541,179.526,5.441,149.094
C08699=1211.672,-83.016,-38.530,179.524,5.440,149.095
C08700=1211.677,-83.266,-38.519,179.522,5.440,149.095
C08701=1211.683,-83.515,-38.508,179.520,5.440,149.096
C08702=1211.688,-83.766,-38.497,179.517,5.440,149.097
C08703=1211.694,-84.015,-38.486,179.515,5.440,149.097
C08704=1211.699,-84.265,-38.476,179.512,5.439,149.098
C08705=1211.704,-84.514,-38.465,179.510,5.440,149.099
C08706=1211.709,-84.764,-38.454,179.508,5.439,149.099
C08707=1211.714,-85.014,-38.443,179.506,5.439,149.100
C08708=1211.720,-85.264,-38.432,179.503,5.439,149.101
C08709=1211.725,-85.514,-38.421,179.501,5.439,149.101
C08710=1211.730,-85.763,-38.410,179.498,5.439,149.102
C08711=1211.735,-86.013,-38.400,179.496,5.438,149.103
C08712=1211.741,-86.262,-38.389,179.494,5.439,149.103
C08713=1211.746,-86.512,-38.378,179.491,5.438,149.104
C08714=1211.751,-86.762,-38.368,179.489,5.438,149.105
C08715=1211.756,-87.011,-38.357,179.487,5.438,149.105
C08716=1211.761,-87.262,-38.346,179.484,5.438,149.106
C08717=1211.766,-87.511,-38.336,179.482,5.438,149.107
C08718=1211.771,-87.761,-38.325,179.480,5.438,149.107
C08719=1211.777,-88.010,-38.315,179.478,5.437,149.108
C08720=1211.782,-88.260,-38.303,179.475,5.438,149.109
C08721=1211.788,-88.510,-38.293,179.473,5.437,149.109
C08722=1211.793,-88.760,-38.282,179.471,5.438,149.110
C08723=1211.798,-89.009,-38.271,179.468,5.437,149.111
C08724=1211.803,-89.259,-38.260,179.466,5.438,149.111
C08725=1211.809,-89.509,-38.250,179.464,5.437,149.112
C08726=1211.813,-89.758,-38.239,179.462,5.437,149.113
C08727=1211.819,-90.008,-38.229,179.459,5.437,149.113
C08728=1211.824,-90.258,-38.218,179.456,5.436,149.114
C08729=1211.830,-90.508,-38.208,179.454,5.437,149.115
C08730=1211.834,-90.757,-38.197,179.452,5.436,149.116
C08731=1211.840,-91.007,-38.186,179.450,5.436,149.116
C08732=1211.845,-91.257,-38.176,179.447,5.436,149.117
C08733=1211.850,-91.507,-38.166,179.445,5.436,149.117
C08734=1211.855,-91.756,-38.154,179.443,5.436,149.118
C08735=1211.861,-92.006,-38.144,179.440,5.436,149.119
C08736=1211.866,-92.256,-38.134,179.438,5.436,149.120
C08737=1211.871,-92.506,-38.123,179.436,5.436,149.120
C08738=1211.876,-92.755,-38.112,179.433,5.435,149.121
C08739=1211.882,-93.005,-38.102,179.431,5.436,149.121
C08740=1211.887,-93.255,-38.091,179.429,5.435,149.122
C08741=1211.892,-93.505,-38.081,179.427,5.436,149.123
C08742=1211.898,-93.754,-38.071,179.424,5.435,149.123
C08743=1211.902,-94.004,-38.060,179.422,5.435,149.124
C08744=1211.908,-94.253,-38.049,179.420,5.435,149.125
C08745=1211.913,-94.503,-38.039,179.418,5.435,149.126
C08746=1211.918,-94.753,-38.029,179.415,5.435,149.126
C08747=1211.923,-95.003,-38.019,179.413,5.435,149.127
C08748=1211.928,-95.252,-38.008,179.411,5.434,149.127
C08749=1211.933,-95.502,-37.997,179.409,5.435,149.128
C08750=1211.939,-95.752,-37.987,179.406,5.434,149.129
C08751=1211.944,-96.001,-37.977,179.404,5.435,149.130
C08752=1211.949,-96.251,-37.966,179.401,5.434,149.130
C08753=1211.955,-96.501,-37.956,179.399,5.433,149.131
C08754=1211.960,-96.751,-37.945,179.397,5.434,149.131
C08755=1211.966,-97.001,-37.935,179.394,5.433,149.132
C08756=1211.971,-97.250,-37.924,179.392,5.434,149.133
C08757=1211.975,-97.500,-37.914,179.389,5.433,149.134
C08758=1211.981,-97.749,-37.904,179.387,5.434,149.134
C08759=1211.986,-97.999,-37.893,179.385,5.433,149.135
C08760=1211.991,-98.249,-37.883,179.383,5.433,149.136
C08761=1211.997,-98.498,-37.873,179.380,5.433,149.136
C08762=1212.002,-98.749,-37.862,179.378,5.433,149.137
C08763=1212.008,-98.998,-37.852,179.376,5.433,149.138
C08764=1212.013,-99.249,-37.842,179.374,5.433,149.138
C08765=1212.017,-99.498,-37.832,179.371,5.432,149.139
C08766=1212.023,-99.747,-37.822,179.369,5.433,149.140
C08767=1212.028,-99.998,-37.811,179.367,5.432,149.140
C08768=1212.034,-100.247,-37.801,179.364,5.433,149.141
C08769=1212.039,-100.497,-37.791,179.362,5.432,149.141
C08770=1212.044,-100.768,-37.780,179.360,5.432,149.142
C08771=1212.050,-101.040,-37.768,179.358,5.432,149.143
C08772=1212.055,-101.311,-37.757,179.355,5.431,149.144
C08773=1212.061,-101.581,-37.747,179.352,5.432,149.145
C08774=1212.066,-101.832,-37.736,179.350,5.431,149.145
C08775=1212.072,-102.081,-37.726,179.348,5.432,149.146
C08776=1212.077,-102.331,-37.716,179.345,5.431,149.146
C08777=1212.082,-102.581,-37.705,179.343,5.432,149.147
C08778=1212.087,-102.830,-37.696,179.341,5.431,149.148
C08779=1212.093,-103.080,-37.685,179.339,5.431,149.148
C08780=1212.098,-103.330,-37.675,179.336,5.431,149.149
C08781=1212.104,-103.580,-37.665,179.334,5.431,149.150
C08782=1212.108,-103.829,-37.655,179.331,5.431,149.151
C08783=1212.113,-104.079,-37.645,179.330,5.431,149.151
C08784=1212.119,-104.329,-37.634,179.327,5.430,149.152
C08785=1212.125,-104.578,-37.624,179.325,5.431,149.152
C08786=1212.129,-104.829,-37.615,179.322,5.430,149.153
C08787=1212.135,-105.078,-37.605,179.320,5.431,149.154
C08788=1212.140,-105.328,-37.594,179.318,5.430,149.154
C08789=1212.146,-105.577,-37.584,179.316,5.430,149.155
C08790=1212.150,-105.827,-37.574,179.313,5.430,149.156
C08791=1212.156,-106.077,-37.564,179.311,5.430,149.156
C08792=1212.161,-106.326,-37.554,179.309,5.430,149.157
C08793=1212.166,-106.576,-37.544,179.307,5.430,149.158
C08794=1212.172,-106.826,-37.534,179.304,5.429,149.158
C08795=1212.177,-107.076,-37.524,179.302,5.430,149.159
C08796=1212.182,-107.325,-37.515,179.300,5.429,149.160
C08797=1212.187,-107.575,-37.504,179.298,5.429,149.160
C08798=1212.193,-107.825,-37.494,179.296,5.430,149.161
C08799=1212.198,-108.075,-37.484,179.293,5.429,149.162
C08800=1212.203,-108.325,-37.474,179.291,5.430,149.162
C08801=1212.208,-108.575,-37.464,179.288,5.429,149.163
C08802=1212.214,-108.824,-37.454,179.287,5.429,149.164
C08803=1212.219,-109.073,-37.444,179.284,5.429,149.164
C08804=1212.224,-109.324,-37.434,179.282,5.429,149.165
C08805=1212.229,-109.574,-37.425,179.279,5.429,149.166
C08806=1212.235,-109.823,-37.415,179.278,5.429,149.166
C08807=1212.240,-110.073,-37.404,179.275,5.428,149.167
C08808=1212.244,-110.323,-37.394,179.273,5.429,149.168
C08809=1212.250,-110.573,-37.385,179.270,5.428,149.168
C08810=1212.256,-110.822,-37.375,179.269,5.428,149.169
C08811=1212.261,-111.071,-37.365,179.266,5.428,149.170
C08812=1212.267,-111.322,-37.356,179.264,5.428,149.170
C08813=1212.271,-111.572,-37.346,179.261,5.428,149.171
C08814=1212.277,-111.821,-37.335,179.260,5.428,149.172
C08815=1212.282,-112.071,-37.325,179.257,5.427,149.172
C08816=1212.287,-112.320,-37.316,179.255,5.428,149.173
C08817=1212.293,-112.570,-37.306,179.252,5.427,149.174
C08818=1212.297,-112.820,-37.296,179.250,5.428,149.174
C08819=1212.303,-113.070,-37.287,179.248,5.427,149.175
C08820=1212.309,-113.320,-37.276,179.246,5.427,149.176
C08821=1212.314,-113.569,-37.267,179.243,5.427,149.176
C08822=1212.319,-113.819,-37.257,179.241,5.427,149.177
C08823=1212.324,-114.069,-37.247,179.239,5.427,149.178
C08824=1212.329,-114.319,-37.237,179.237,5.427,149.178
C08825=1212.334,-114.568,-37.228,179.235,5.427,149.179
C08826=1212.340,-114.818,-37.218,179.232,5.427,149.180
C08827=1212.346,-115.067,-37.208,179.230,5.427,149.180
C08828=1212.351,-115.317,-37.199,179.228,5.427,149.181
C08829=1212.356,-115.568,-37.188,179.226,5.427,149.182
C08830=1212.361,-115.817,-37.179,179.223,5.427,149.182
C08831=1212.367,-116.067,-37.169,179.221,5.427,149.183
C08832=1212.371,-116.316,-37.160,179.219,5.426,149.183
C08833=1212.377,-116.566,-37.150,179.217,5.427,149.184
C08834=1212.382,-116.816,-37.140,179.214,5.426,149.185
C08835=1212.388,-117.066,-37.131,179.212,5.426,149.185
C08836=1212.392,-117.316,-37.121,179.210,5.426,149.186
C08837=1212.398,-117.566,-37.112,179.208,5.426,149.187
C08838=1212.403,-117.815,-37.102,179.205,5.425,149.187
C08839=1212.409,-118.065,-37.092,179.203,5.426,149.188
C08840=1212.414,-118.314,-37.083,179.201,5.425,149.189
C08841=1212.420,-118.564,-37.073,179.199,5.426,149.189
C08842=1212.424,-118.815,-37.063,179.197,5.426,149.190
C08843=1212.430,-119.064,-37.053,179.194,5.425,149.191
C08844=1212.435,-119.314,-37.044,179.192,5.426,149.191
C08845=1212.440,-119.563,-37.035,179.190,5.425,149.192
C08846=1212.446,-119.813,-37.025,179.188,5.425,149.193
C08847=1212.450,-120.063,-37.015,179.185,5.425,149.193
C08848=1212.456,-120.313,-37.006,179.183,5.425,149.194
C08849=1212.461,-120.562,-36.996,179.180,5.425,149.195
C08850=1212.467,-120.812,-36.987,179.179,5.425,149.195
C08851=1212.471,-121.062,-36.977,179.176,5.424,149.196
C08852=1212.477,-121.312,-36.967,179.174,5.425,149.197
C08853=1212.482,-121.562,-36.959,179.172,5.424,149.197
C08854=1212.487,-121.811,-36.949,179.170,5.424,149.198
C08855=1212.493,-122.062,-36.939,179.167,5.424,149.199
C08856=1212.498,-122.311,-36.930,179.165,5.424,149.199
C08857=1212.504,-122.561,-36.920,179.163,5.424,149.200
C08858=1212.509,-122.810,-36.911,179.161,5.424,149.200
C08859=1212.514,-123.060,-36.902,179.159,5.424,149.201
C08860=1212.520,-123.310,-36.892,179.156,5.424,149.202
C08861=1212.525,-123.559,-36.883,179.154,5.424,149.202
C08862=1212.530,-123.809,-36.874,179.152,5.424,149.203
C08863=1212.536,-124.059,-36.864,179.150,5.424,149.204
C08864=1212.540,-124.309,-36.854,179.147,5.423,149.204
C08865=1212.546,-124.559,-36.845,179.145,5.424,149.205
C08866=1212.551,-124.809,-36.835,179.143,5.423,149.206
C08867=1212.556,-125.059,-36.826,179.141,5.423,149.206
C08868=1212.562,-125.308,-36.816,179.139,5.424,149.207
C08869=1212.567,-125.558,-36.807,179.136,5.423,149.208
C08870=1212.572,-125.808,-36.798,179.134,5.424,149.208
C08871=1212.578,-126.057,-36.788,179.132,5.423,149.209
C08872=1212.583,-126.307,-36.779,179.130,5.423,149.210
C08873=1212.588,-126.557,-36.770,179.127,5.423,149.210
C08874=1212.167,-126.568,-36.808,179.123,5.426,149.212
C08875=1212.162,-126.318,-36.817,179.126,5.426,149.211
C08876=1212.156,-126.068,-36.826,179.128,5.426,149.211
C08877=1212.151,-125.818,-36.836,179.130,5.427,149.210
C08878=1212.146,-125.569,-36.845,179.132,5.426,149.210
C08879=1212.140,-125.318,-36.854,179.135,5.427,149.209
C08880=1212.135,-125.069,-36.864,179.137,5.427,149.208
C08881=1212.130,-124.819,-36.873,179.139,5.426,149.208
C08882=1212.124,-124.569,-36.882,179.141,5.427,149.207
C08883=1212.119,-124.320,-36.892,179.143,5.427,149.206
C08884=1212.114,-124.070,-36.901,179.146,5.427,149.206
C08885=1212.108,-123.820,-36.910,179.148,5.427,149.205
C08886=1212.103,-123.571,-36.920,179.150,5.428,149.205
C08887=1212.097,-123.321,-36.929,179.152,5.427,149.204
C08888=1212.093,-123.071,-36.939,179.155,5.428,149.203
C08889=1212.087,-122.822,-36.948,179.157,5.427,149.202
C08890=1212.082,-122.571,-36.957,179.159,5.428,149.202
C08891=1212.077,-122.322,-36.967,179.161,5.428,149.201
C08892=1212.071,-122.071,-36.977,179.163,5.427,149.200
C08893=1212.067,-121.822,-36.986,179.165,5.428,149.200
C08894=1212.061,-121.572,-36.995,179.167,5.428,149.199
C08895=1212.056,-121.323,-37.005,179.170,5.428,149.199
C08896=1212.051,-121.073,-37.014,179.172,5.428,149.198
C08897=1212.045,-120.823,-37.025,179.174,5.428,149.197
C08898=1212.040,-120.573,-37.033,179.177,5.428,149.197
C08899=1212.035,-120.324,-37.042,179.179,5.428,149.196
C08900=1212.029,-120.074,-37.053,179.181,5.428,149.195
C08901=1212.024,-119.824,-37.061,179.183,5.429,149.195
C08902=1212.018,-119.575,-37.072,179.186,5.428,149.194
C08903=1212.014,-119.324,-37.081,179.188,5.429,149.193
C08904=1212.008,-119.074,-37.091,179.190,5.429,149.193
C08905=1212.003,-118.825,-37.100,179.193,5.429,149.192
C08906=1211.997,-118.575,-37.110,179.195,5.429,149.191
C08907=1211.992,-118.326,-37.120,179.197,5.428,149.191
C08908=1211.987,-118.076,-37.129,179.199,5.429,149.190
C08909=1211.982,-117.826,-37.139,179.201,5.429,149.189
C08910=1211.977,-117.577,-37.148,179.204,5.429,149.189
C08911=1211.972,-117.326,-37.158,179.205,5.429,149.188
C08912=1211.966,-117.077,-37.167,179.208,5.430,149.187
C08913=1211.961,-116.827,-37.178,179.210,5.429,149.187
C08914=1211.956,-116.577,-37.186,179.213,5.430,149.186
C08915=1211.950,-116.328,-37.197,179.214,5.430,149.186
C08916=1211.945,-116.078,-37.206,179.217,5.430,149.185
C08917=1211.940,-115.827,-37.216,179.219,5.430,149.184
C08918=1211.934,-115.578,-37.226,179.222,5.430,149.183
C08919=1211.929,-115.328,-37.235,179.223,5.430,149.183
C08920=1211.924,-115.079,-37.245,179.226,5.431,149.182
C08921=1211.919,-114.829,-37.255,179.228,5.430,149.182
C08922=1211.913,-114.579,-37.265,179.231,5.431,149.181
C08923=1211.908,-114.329,-37.275,179.232,5.431,149.180
C08924=1211.903,-114.079,-37.284,179.235,5.430,149.180
C08925=1211.898,-113.830,-37.294,179.237,5.431,149.179
C08926=1211.892,-113.580,-37.304,179.239,5.430,149.178
C08927=1211.887,-113.330,-37.313,179.241,5.431,149.178
C08928=1211.881,-113.081,-37.323,179.244,5.431,149.177
C08929=1211.876,-112.831,-37.334,179.246,5.431,149.176
C08930=1211.871,-112.581,-37.342,179.248,5.431,149.176
C08931=1211.866,-112.331,-37.353,179.251,5.431,149.175
C08932=1211.861,-112.082,-37.362,179.253,5.431,149.174
C08933=1211.855,-111.832,-37.372,179.255,5.431,149.174
C08934=1211.850,-111.582,-37.382,179.257,5.431,149.173
C08935=1211.845,-111.332,-37.392,179.260,5.432,149.172
C08936=1211.839,-111.083,-37.402,179.262,5.431,149.172
C08937=1211.834,-110.833,-37.411,179.264,5.432,149.171
C08938=1211.829,-110.583,-37.422,179.266,5.432,149.170
C08939=1211.824,-110.333,-37.432,179.269,5.432,149.170
C08940=1211.819,-110.084,-37.441,179.271,5.432,149.169
C08941=1211.813,-109.834,-37.451,179.273,5.432,149.168
C08942=1211.807,-109.584,-37.461,179.275,5.432,149.168
C08943=1211.803,-109.334,-37.471,179.278,5.432,149.167
C08944=1211.797,-109.085,-37.481,179.280,5.432,149.166
C08945=1211.791,-108.835,-37.491,179.282,5.433,149.166
C08946=1211.787,-108.585,-37.500,179.285,5.432,149.165
C08947=1211.782,-108.335,-37.511,179.287,5.433,149.164
C08948=1211.776,-108.086,-37.521,179.289,5.433,149.164
C08949=1211.771,-107.836,-37.531,179.291,5.433,149.163
C08950=1211.765,-107.586,-37.540,179.294,5.433,149.162
C08951=1211.760,-107.336,-37.551,179.296,5.433,149.162
C08952=1211.755,-107.087,-37.560,179.298,5.433,149.161
C08953=1211.750,-106.837,-37.571,179.300,5.433,149.160
C08954=1211.745,-106.587,-37.581,179.303,5.433,149.160
C08955=1211.740,-106.338,-37.591,179.305,5.433,149.159
C08956=1211.734,-106.088,-37.600,179.307,5.433,149.158
C08957=1211.728,-105.838,-37.611,179.309,5.433,149.158
C08958=1211.724,-105.588,-37.621,179.312,5.434,149.157
C08959=1211.719,-105.339,-37.631,179.314,5.433,149.156
C08960=1211.713,-105.089,-37.641,179.316,5.434,149.156
C08961=1211.708,-104.839,-37.652,179.318,5.434,149.155
C08962=1211.703,-104.589,-37.661,179.321,5.434,149.155
C08963=1211.698,-104.340,-37.671,179.323,5.434,149.154
C08964=1211.692,-104.089,-37.681,179.325,5.434,149.153
C08965=1211.687,-103.840,-37.691,179.328,5.434,149.152
C08966=1211.682,-103.590,-37.701,179.330,5.435,149.152
C08967=1211.677,-103.340,-37.712,179.332,5.434,149.151
C08968=1211.671,-103.091,-37.722,179.334,5.435,149.150
C08969=1211.666,-102.841,-37.732,179.337,5.434,149.150
C08970=1211.661,-102.592,-37.742,179.339,5.435,149.149
C08971=1211.656,-102.342,-37.752,179.341,5.435,149.149
C08972=1211.650,-102.092,-37.762,179.344,5.435,149.148
C08973=1211.645,-101.842,-37.773,179.346,5.435,149.147
C08974=1211.640,-101.592,-37.783,179.348,5.435,149.146
C08975=1211.634,-101.321,-37.794,179.351,5.436,149.146
C08976=1211.629,-101.050,-37.805,179.353,5.435,149.145
C08977=1211.623,-100.779,-37.816,179.356,5.436,149.144
C08978=1211.617,-100.507,-37.827,179.358,5.435,149.144
C08979=1211.612,-100.258,-37.837,179.361,5.436,149.143
C08980=1211.606,-100.008,-37.848,179.362,5.436,149.142
C08981=1211.601,-99.758,-37.858,179.365,5.436,149.142
C08982=1211.596,-99.509,-37.868,179.367,5.436,149.141
C08983=1211.591,-99.259,-37.878,179.370,5.436,149.140
C08984=1211.586,-99.009,-37.889,179.372,5.436,149.140
C08985=1211.580,-98.759,-37.899,179.374,5.437,149.139
C08986=1211.575,-98.509,-37.909,179.376,5.436,149.138
C08987=1211.570,-98.260,-37.920,179.379,5.437,149.138
C08988=1211.564,-98.010,-37.930,179.381,5.436,149.137
C08989=1211.560,-97.760,-37.940,179.383,5.437,149.136
C08990=1211.554,-97.511,-37.950,179.386,5.438,149.136
C08991=1211.549,-97.261,-37.961,179.388,5.437,149.135
C08992=1211.544,-97.012,-37.972,179.390,5.438,149.134
C08993=1211.538,-96.762,-37.982,179.392,5.437,149.134
C08994=1211.533,-96.512,-37.992,179.395,5.438,149.133
C08995=1211.528,-96.262,-38.003,179.397,5.437,149.132
C08996=1211.523,-96.012,-38.013,179.399,5.438,149.132
C08997=1211.517,-95.762,-38.023,179.401,5.438,149.131
C08998=1211.512,-95.512,-38.034,179.404,5.438,149.130
C08999=1211.507,-95.263,-38.043,179.406,5.438,149.130
C09000=1211.502,-95.014,-38.054,179.409,5.438,149.129
C09001=1211.497,-94.764,-38.065,179.410,5.438,149.128
C09002=1211.491,-94.514,-38.075,179.413,5.439,149.128
C09003=1211.486,-94.264,-38.086,179.415,5.438,149.127
C09004=1211.481,-94.014,-38.096,179.418,5.439,149.126
C09005=1211.476,-93.764,-38.107,179.420,5.438,149.125
C09006=1211.470,-93.515,-38.117,179.422,5.439,149.125
C09007=1211.465,-93.266,-38.128,179.424,5.439,149.124
C09008=1211.460,-93.015,-38.138,179.427,5.439,149.124
C09009=1211.454,-92.766,-38.148,179.429,5.439,149.123
C09010=1211.449,-92.516,-38.159,179.432,5.439,149.122
C09011=1211.444,-92.267,-38.170,179.434,5.439,149.121
C09012=1211.439,-92.016,-38.181,179.436,5.440,149.121
C09013=1211.433,-91.767,-38.191,179.438,5.439,149.120
C09014=1211.428,-91.517,-38.201,179.441,5.440,149.120
C09015=1211.423,-91.268,-38.212,179.443,5.439,149.119
C09016=1211.418,-91.018,-38.223,179.446,5.440,149.118
C09017=1211.412,-90.768,-38.233,179.448,5.439,149.117
C09018=1211.407,-90.518,-38.244,179.450,5.440,149.117
C09019=1211.402,-90.269,-38.255,179.452,5.441,149.116
C09020=1211.397,-90.019,-38.265,179.455,5.440,149.115
C09021=1211.392,-89.769,-38.275,179.457,5.441,149.115
C09022=1211.387,-89.519,-38.287,179.459,5.440,149.114
C09023=1211.381,-89.270,-38.297,179.461,5.441,149.114
C09024=1211.376,-89.020,-38.307,179.464,5.441,149.113
C09025=1211.371,-88.771,-38.318,179.466,5.441,149.112
C09026=1211.366,-88.520,-38.329,179.468,5.441,149.111
C09027=1211.360,-88.271,-38.339,179.471,5.441,149.111
C09028=1211.356,-88.021,-38.350,179.473,5.441,149.110
C09029=1211.350,-87.772,-38.361,179.475,5.442,149.110
C09030=1211.345,-87.522,-38.371,179.477,5.441,149.109
C09031=1211.340,-87.273,-38.382,179.480,5.442,149.108
C09032=1211.335,-87.022,-38.393,179.482,5.441,149.107
C09033=1211.328,-86.772,-38.403,179.485,5.442,149.107
C09034=1211.324,-86.523,-38.415,179.487,5.442,149.106
C09035=1211.319,-86.273,-38.425,179.490,5.442,149.105
C09036=1211.313,-86.024,-38.436,179.492,5.443,149.105
C09037=1211.308,-85.773,-38.447,179.494,5.442,149.104
C09038=1211.303,-85.524,-38.457,179.497,5.443,149.103
C09039=1211.298,-85.274,-38.468,179.499,5.442,149.103
C09040=1211.293,-85.025,-38.479,179.501,5.443,149.102
C09041=1211.288,-84.775,-38.490,179.503,5.442,149.101
C09042=1211.282,-84.526,-38.500,179.506,5.443,149.101
C09043=1211.277,-84.276,-38.512,179.508,5.443,149.100
C09044=1211.272,-84.025,-38.522,179.510,5.443,149.099
C09045=1211.266,-83.776,-38.533,179.512,5.443,149.099
C09046=1211.262,-83.526,-38.544,179.515,5.443,149.098
C09047=1211.256,-83.277,-38.554,179.518,5.444,149.097
C09048=1211.251,-83.027,-38.565,179.519,5.444,149.097
C09049=1211.246,-82.777,-38.576,179.522,5.444,149.096
C09050=1211.240,-82.528,-38.588,179.524,5.444,149.095
C09051=1211.235,-82.277,-38.598,179.527,5.444,149.095
C09052=1211.230,-82.028,-38.609,179.529,5.444,149.094
C09053=1211.225,-81.778,-38.620,179.532,5.444,149.093
C09054=1211.220,-81.529,-38.631,179.534,5.444,149.092
C09055=1211.214,-81.279,-38.642,179.536,5.445,149.092
C09056=1211.209,-81.029,-38.653,179.538,5.445,149.091
C09057=1211.204,-80.780,-38.664,179.541,5.445,149.091
C09058=1211.199,-80.530,-38.675,179.543,5.445,149.090
C09059=1211.194,-80.280,-38.686,179.545,5.445,149.089
C09060=1211.188,-80.030,-38.697,179.548,5.446,149.088
C09061=1211.183,-79.781,-38.708,179.550,5.445,149.088
C09062=1211.178,-79.531,-38.718,179.552,5.446,149.087
C09063=1211.173,-79.282,-38.729,179.554,5.446,149.087
C09064=1211.168,-79.032,-38.741,179.557,5.446,149.086
C09065=1211.163,-78.781,-38.752,179.559,5.446,149.085
C09066=1211.157,-78.532,-38.763,179.562,5.446,149.084
C09067=1211.152,-78.282,-38.773,179.564,5.447,149.084
C09068=1211.146,-78.033,-38.785,179.567,5.446,149.083
C09069=1211.142,-77.783,-38.796,179.569,5.447,149.083
C09070=1211.137,-77.533,-38.807,179.571,5.447,149.082
C09071=1211.131,-77.284,-38.818,179.573,5.447,149.081
C09072=1211.126,-77.034,-38.829,179.576,5.447,149.080
C09073=1211.121,-76.784,-38.840,179.578,5.447,149.080
C09074=1211.116,-76.535,-38.851,179.580,5.447,149.079
C09075=1211.110,-76.285,-38.862,179.583,5.447,149.078
C09076=1211.105,-76.035,-38.874,179.585,5.448,149.078
C09077=1211.100,-75.786,-38.884,179.587,5.448,149.077
C09078=1211.095,-75.536,-38.895,179.590,5.448,149.076
C09079=1211.090,-75.265,-38.908,179.592,5.448,149.076
C09080=1211.083,-74.995,-38.920,179.595,5.448,149.075
C09081=1211.078,-74.724,-38.932,179.597,5.449,149.074
C09082=1211.072,-74.453,-38.944,179.600,5.448,149.073
C09083=1211.067,-74.204,-38.955,179.602,5.449,149.073
C09084=1211.062,-73.954,-38.966,179.605,5.449,149.072
C09085=1211.056,-73.704,-38.978,179.607,5.449,149.071
C09086=1211.052,-73.454,-38.989,179.610,5.449,149.071
C09087=1211.046,-73.206,-39.000,179.612,5.449,149.070
C09088=1211.041,-72.955,-39.011,179.614,5.449,149.069
C09089=1211.036,-72.705,-39.022,179.616,5.449,149.069
C09090=1211.030,-72.456,-39.034,179.619,5.450,149.068
C09091=1211.025,-72.206,-39.045,179.621,5.450,149.067
C09092=1211.021,-71.957,-39.057,179.623,5.450,149.067
C09093=1211.015,-71.706,-39.068,179.626,5.450,149.066
C09094=1211.009,-71.457,-39.079,179.628,5.450,149.065
C09095=1211.004,-71.207,-39.091,179.631,5.450,149.065
C09096=1210.999,-70.958,-39.102,179.633,5.450,149.064
C09097=1210.995,-70.708,-39.113,179.636,5.451,149.063
C09098=1210.988,-70.458,-39.124,179.638,5.451,149.063
C09099=1210.984,-70.209,-39.135,179.640,5.451,149.062
C09100=1210.978,-69.959,-39.147,179.642,5.451,149.061
C09101=1210.974,-69.709,-39.158,179.645,5.451,149.061
C09102=1210.967,-69.460,-39.170,179.647,5.452,149.060
C09103=1210.963,-69.210,-39.181,179.650,5.452,149.059
C09104=1210.958,-68.961,-39.192,179.652,5.452,149.058
C09105=1210.952,-68.710,-39.204,179.655,5.452,149.058
C09106=1210.948,-68.460,-39.215,179.656,5.452,149.057
C09107=1210.942,-68.211,-39.226,179.659,5.453,149.057
C09108=1210.937,-67.962,-39.238,179.661,5.452,149.056
C09109=1210.932,-67.712,-39.250,179.664,5.453,149.055
C09110=1210.927,-67.462,-39.261,179.666,5.453,149.054
C09111=1210.921,-67.212,-39.273,179.668,5.453,149.054
C09112=1210.916,-66.963,-39.284,179.671,5.453,149.053
C09113=1210.911,-66.713,-39.296,179.673,5.453,149.052
C09114=1210.906,-66.464,-39.307,179.675,5.454,149.052
C09115=1210.901,-66.214,-39.319,179.678,5.454,149.051
C09116=1210.896,-65.964,-39.330,179.680,5.454,149.050
C09117=1210.890,-65.715,-39.342,179.683,5.454,149.050
C09118=1210.885,-65.465,-39.353,179.685,5.454,149.049
C09119=1210.879,-65.215,-39.364,179.688,5.454,149.048
C09120=1210.875,-64.965,-39.375,179.690,5.455,149.048
C09121=1210.869,-64.715,-39.387,179.692,5.454,149.047
C09122=1210.865,-64.465,-39.399,179.694,5.455,149.046
C09123=1210.859,-64.216,-39.410,179.697,5.455,149.046
C09124=1210.854,-63.967,-39.422,179.699,5.455,149.045
C09125=1210.849,-63.717,-39.434,179.702,5.456,149.044
C09126=1210.844,-63.468,-39.445,179.704,5.455,149.044
C09127=1210.839,-63.218,-39.457,179.707,5.456,149.043
C09128=1210.833,-62.968,-39.469,179.709,5.455,149.042
C09129=1210.829,-62.718,-39.480,179.711,5.456,149.041
C09130=1210.822,-62.469,-39.492,179.714,5.456,149.041
C09131=1210.818,-62.219,-39.503,179.716,5.456,149.040
C09132=1210.812,-61.969,-39.515,179.718,5.457,149.040
C09133=1210.808,-61.720,-39.526,179.720,5.457,149.039
C09134=1210.802,-61.470,-39.538,179.723,5.457,149.038
C09135=1210.797,-61.220,-39.550,179.726,5.457,149.037
C09136=1210.792,-60.970,-39.561,179.728,5.457,149.037
C09137=1210.787,-60.720,-39.573,179.730,5.458,149.036
C09138=1210.781,-60.471,-39.584,179.733,5.457,149.035
